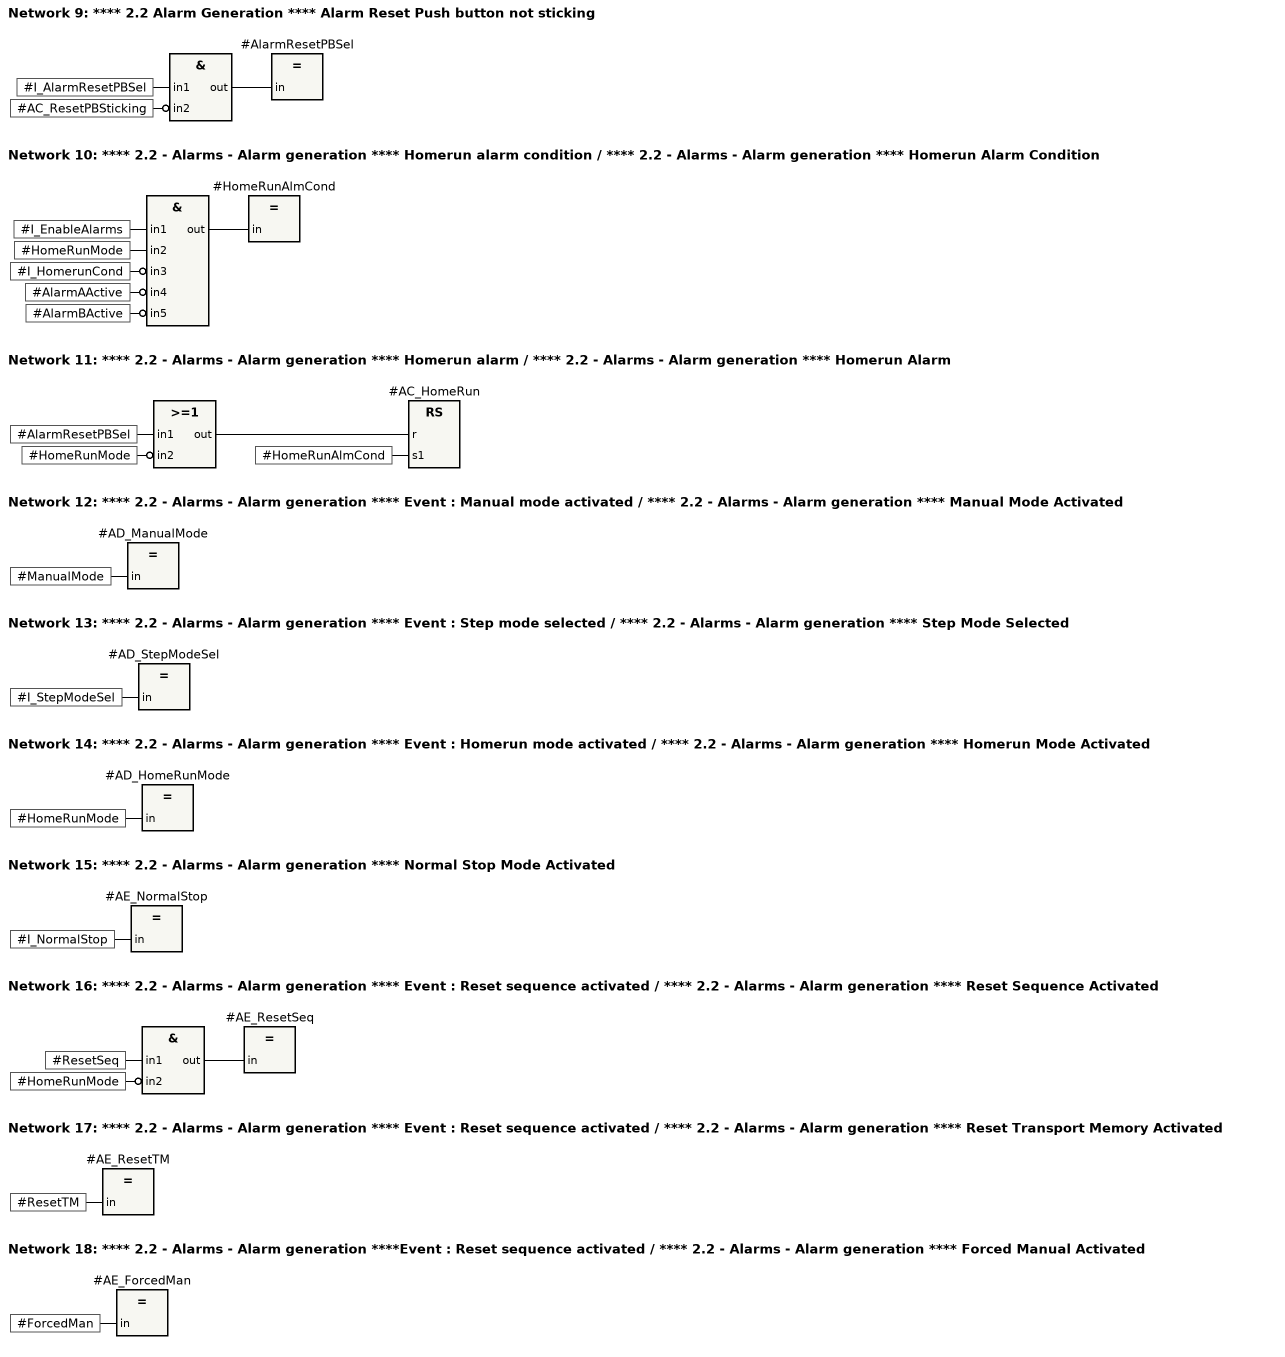
   #AlarmResetPBSel := #I_AlarmResetPBSel AND NOT #AC_ResetPBSticking;
END_REGION

REGION Network 10: **** 2.2 - Alarms - Alarm generation **** Homerun alarm condition / **** 2.2 - Alarms - Alarm generation **** Homerun Alarm Condition
   // Homerun alarm condition
   #HomeRunAlmCond := #I_EnableAlarms AND #HomeRunMode AND NOT #I_HomerunCond AND NOT #AlarmAActive AND NOT #AlarmBActive;
END_REGION

REGION Network 11: **** 2.2 - Alarms - Alarm generation **** Homerun alarm / **** 2.2 - Alarms - Alarm generation **** Homerun Alarm
   // Homerun alarm
   IF #AlarmResetPBSel OR NOT #HomeRunMode THEN
       #AC_HomeRun := FALSE;   // RS flip-flop
   END_IF;
   IF #HomeRunAlmCond THEN #AC_HomeRun := TRUE; END_IF;
END_REGION

REGION Network 12: **** 2.2 - Alarms - Alarm generation **** Event : Manual mode activated / **** 2.2 - Alarms - Alarm generation **** Manual Mode Activated
   // Event : Manual mode activated / Event : Manual Mode activated
   #AD_ManualMode := #ManualMode;
END_REGION

REGION Network 13: **** 2.2 - Alarms - Alarm generation **** Event : Step mode selected / **** 2.2 - Alarms - Alarm generation **** Step Mode Selected
   // Event : Step mode selected / Event : Step Mode selected
   #AD_StepModeSel := #I_StepModeSel;
END_REGION

REGION Network 14: **** 2.2 - Alarms - Alarm generation **** Event : Homerun mode activated / **** 2.2 - Alarms - Alarm generation **** Homerun Mode Activated
   // Event : Homerun mode activated / Event : Homerun Mode activated
   #AD_HomeRunMode := #HomeRunMode;
END_REGION

REGION Network 15: **** 2.2 - Alarms - Alarm generation **** Normal Stop Mode Activated
   // Event : Normal Stop Mode activated
   #AE_NormalStop := #I_NormalStop;
END_REGION

REGION Network 16: **** 2.2 - Alarms - Alarm generation **** Event : Reset sequence activated / **** 2.2 - Alarms - Alarm generation **** Reset Sequence Activated
   // Event : Reset sequence activated
   #AE_ResetSeq := #ResetSeq AND NOT #HomeRunMode;
END_REGION

REGION Network 17: **** 2.2 - Alarms - Alarm generation **** Event : Reset sequence activated / **** 2.2 - Alarms - Alarm generation **** Reset Transport Memory Activated
   // Event : Reset sequence activated / Event : Reset transport memory activated
   #AE_ResetTM := #ResetTM;
END_REGION

REGION Network 18: **** 2.2 - Alarms - Alarm generation ****Event : Reset sequence activated / **** 2.2 - Alarms - Alarm generation **** Forced Manual Activated
   // Event : Reset sequence activated / Event : Forced manual activated
   #AE_ForcedMan := #ForcedMan;
END_REGION

REGION Network 19: **** 2.2 - Alarms - Alarm generation **** Auto selected, but not started / **** 2.2 - Alarms - Alarm generation **** Auto Selected, But not Started
   // Auto selected, but not started
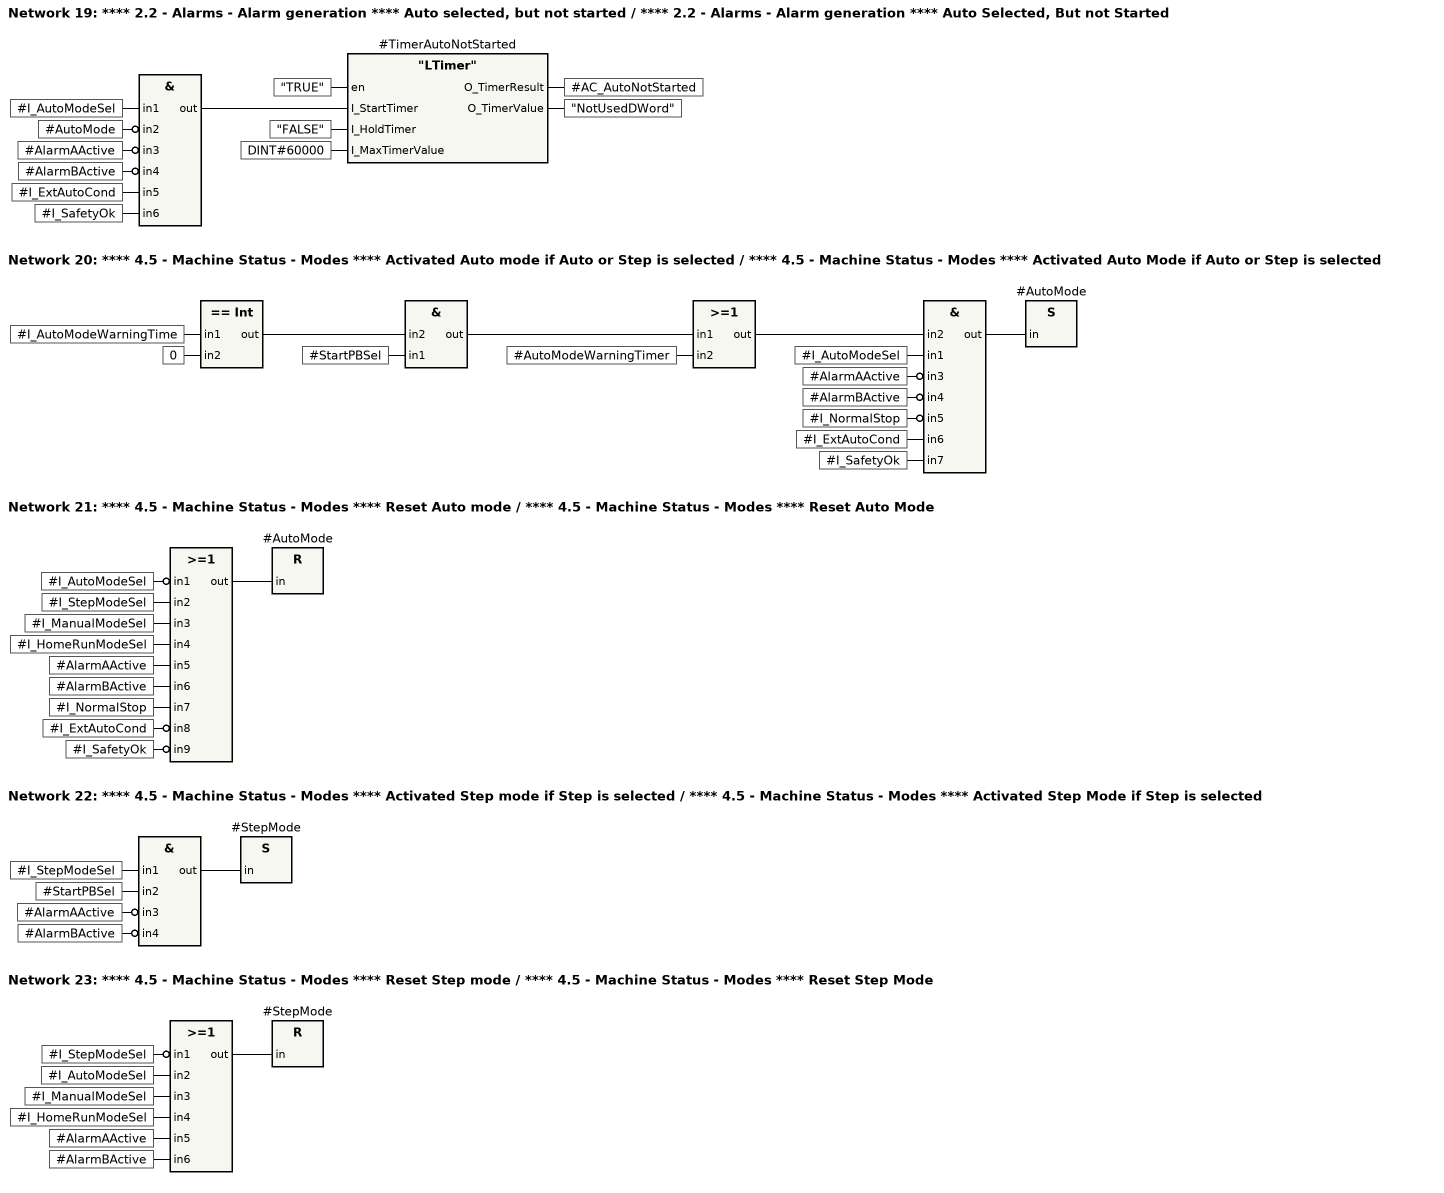
   IF "TRUE" THEN
       #TimerAutoNotStarted(I_StartTimer := #I_AutoModeSel AND NOT #AutoMode AND NOT #AlarmAActive AND NOT #AlarmBActive AND #I_ExtAutoCond AND #I_SafetyOk,   // "LTimer"
                            I_HoldTimer := "FALSE",
                            I_MaxTimerValue := DINT#60000,
                            O_TimerResult => #AC_AutoNotStarted,
                            O_TimerValue => "NotUsedDWord");
   END_IF;
END_REGION

REGION Network 20: **** 4.5 - Machine Status - Modes **** Activated Auto mode if Auto or Step is selected / **** 4.5 - Machine Status - Modes **** Activated Auto Mode if Auto or Step is selected
   // Activated Auto mode if Auto or Step is selected / Activated Auto Mode if Auto or Step is selected
   IF (((#I_AutoModeWarningTime = 0) AND #StartPBSel) OR #AutoModeWarningTimer) AND #I_AutoModeSel AND NOT #AlarmAActive AND NOT #AlarmBActive AND NOT #I_NormalStop AND #I_ExtAutoCond AND #I_SafetyOk THEN
       #AutoMode := TRUE;
   END_IF;
END_REGION

REGION Network 21: **** 4.5 - Machine Status - Modes **** Reset Auto mode / **** 4.5 - Machine Status - Modes **** Reset Auto Mode
   // Reset Auto mode / Reset Auto Mode
   IF NOT #I_AutoModeSel OR #I_StepModeSel OR #I_ManualModeSel OR #I_HomeRunModeSel OR #AlarmAActive OR #AlarmBActive OR #I_NormalStop OR NOT #I_ExtAutoCond OR NOT #I_SafetyOk THEN
       #AutoMode := FALSE;
   END_IF;
END_REGION

REGION Network 22: **** 4.5 - Machine Status - Modes **** Activated Step mode if Step is selected / **** 4.5 - Machine Status - Modes **** Activated Step Mode if Step is selected
   // Activated Step mode if Step is selected / Activated Step Mode if Step is selected
   IF #I_StepModeSel AND #StartPBSel AND NOT #AlarmAActive AND NOT #AlarmBActive THEN
       #StepMode := TRUE;
   END_IF;
END_REGION

REGION Network 23: **** 4.5 - Machine Status - Modes **** Reset Step mode / **** 4.5 - Machine Status - Modes **** Reset Step Mode
   // Reset Step mode / Reset Step Mode
   IF NOT #I_StepModeSel OR #I_AutoModeSel OR #I_ManualModeSel OR #I_HomeRunModeSel OR #AlarmAActive OR #AlarmBActive THEN
       #StepMode := FALSE;
   END_IF;
END_REGION

REGION Network 24: **** 4.5 - Machine Status - Modes **** Activate Homerun mode if all robots are out of station / **** 4.5 - Machine Status - Modes **** Activate Homerun Mode if all robots are out of station
   // Activate Homerun mode if all robots are out of station / Activate Homerun Mode if all robots are out of station
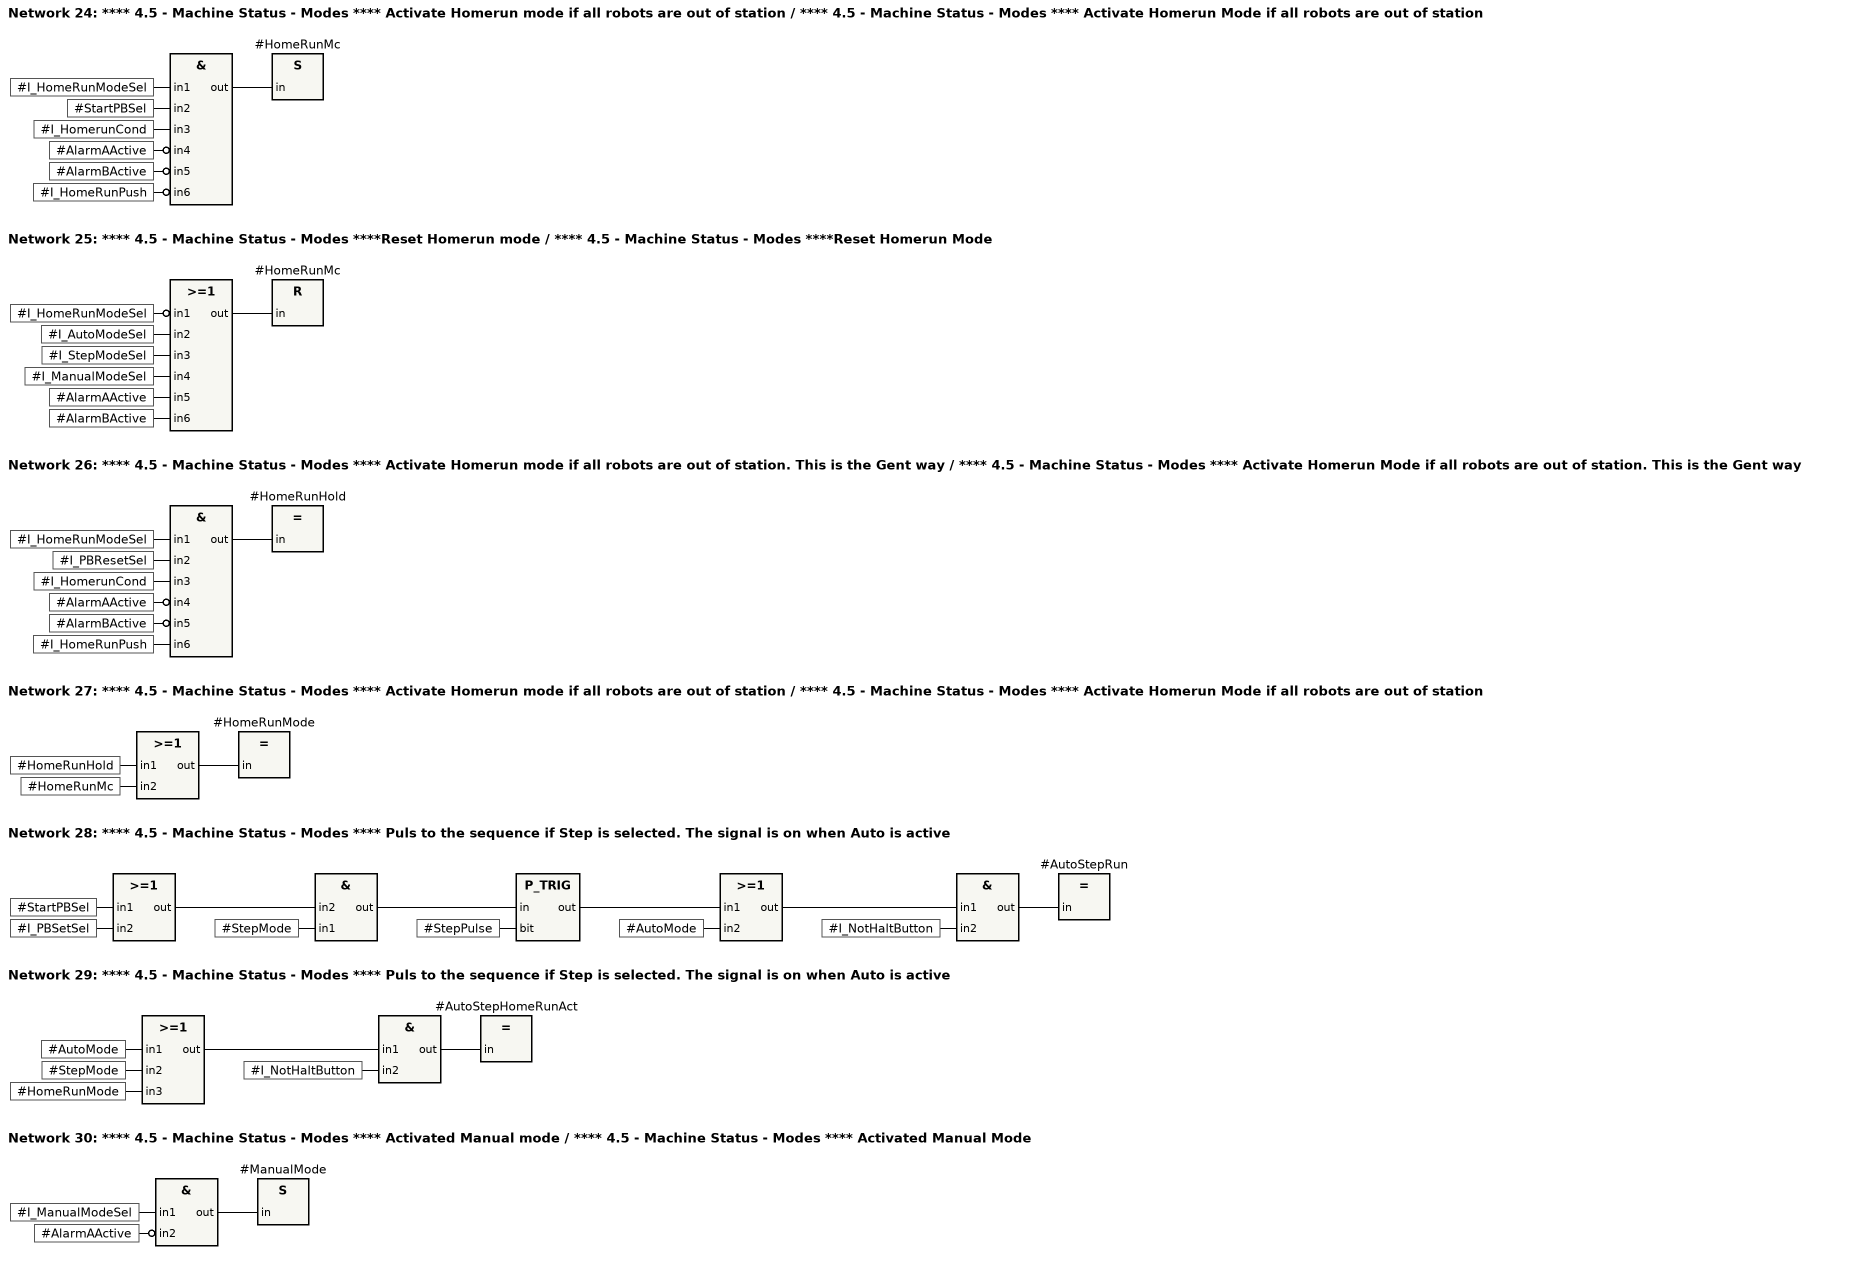
   IF #I_HomeRunModeSel AND #StartPBSel AND #I_HomerunCond AND NOT #AlarmAActive AND NOT #AlarmBActive AND NOT #I_HomeRunPush THEN
       #HomeRunMc := TRUE;
   END_IF;
END_REGION

REGION Network 25: **** 4.5 - Machine Status - Modes ****Reset Homerun mode / **** 4.5 - Machine Status - Modes ****Reset Homerun Mode
   // Reset Homerun mode / Reset Homerun Mode
   IF NOT #I_HomeRunModeSel OR #I_AutoModeSel OR #I_StepModeSel OR #I_ManualModeSel OR #AlarmAActive OR #AlarmBActive THEN
       #HomeRunMc := FALSE;
   END_IF;
END_REGION

REGION Network 26: **** 4.5 - Machine Status - Modes **** Activate Homerun mode if all robots are out of station. This is the Gent way / **** 4.5 - Machine Status - Modes **** Activate Homerun Mode if all robots are out of station. This is the Gent way
   // Activate Homerun mode if all robots are out of station. This is the Gent way 
   // there the reset pushbutton have to be pressed during the complete homerun.
   // Activate Homerun Mode if all robots are out of station. This is the Gent way 
   // there the reset pushbutton have to be pressed during the complete homerun.
   #HomeRunHold := #I_HomeRunModeSel AND #I_PBResetSel AND #I_HomerunCond AND NOT #AlarmAActive AND NOT #AlarmBActive AND #I_HomeRunPush;
END_REGION

REGION Network 27: **** 4.5 - Machine Status - Modes **** Activate Homerun mode if all robots are out of station / **** 4.5 - Machine Status - Modes **** Activate Homerun Mode if all robots are out of station
   // Activate Homerun mode if all robots are out of station. / Activate Homerun Mode if all robots are out of station.
   #HomeRunMode := #HomeRunHold OR #HomeRunMc;
END_REGION

REGION Network 28: **** 4.5 - Machine Status - Modes **** Puls to the sequence if Step is selected. The signal is on when Auto is active
   // Puls to the sequence if Step is selected. The signal is on when Auto is active.
   #_w1 := (#StartPBSel OR #I_PBSetSel) AND #StepMode;
   #_w2 := #_w1 AND NOT #StepPulse;   // rising edge
   #StepPulse := #_w1;
   #AutoStepRun := (#_w2 OR #AutoMode) AND #I_NotHaltButton;
END_REGION

REGION Network 29: **** 4.5 - Machine Status - Modes **** Puls to the sequence if Step is selected. The signal is on when Auto is active
   // Puls to the sequence if Step is selected. The signal is on when Auto is active.
   #AutoStepHomeRunAct := (#AutoMode OR #StepMode OR #HomeRunMode) AND #I_NotHaltButton;
END_REGION

REGION Network 30: **** 4.5 - Machine Status - Modes **** Activated Manual mode / **** 4.5 - Machine Status - Modes **** Activated Manual Mode
   // Activated Manual mode / Activated Manual Mode
   IF #I_ManualModeSel AND NOT #AlarmAActive THEN #ManualMode := TRUE; END_IF;
END_REGION

REGION Network 31: **** 4.5 - Machine Status - Modes **** Reset Manual mode / **** 4.5 - Machine Status - Modes **** Reset Manual Mode
   // Reset Manual mode / Reset Manual Mode
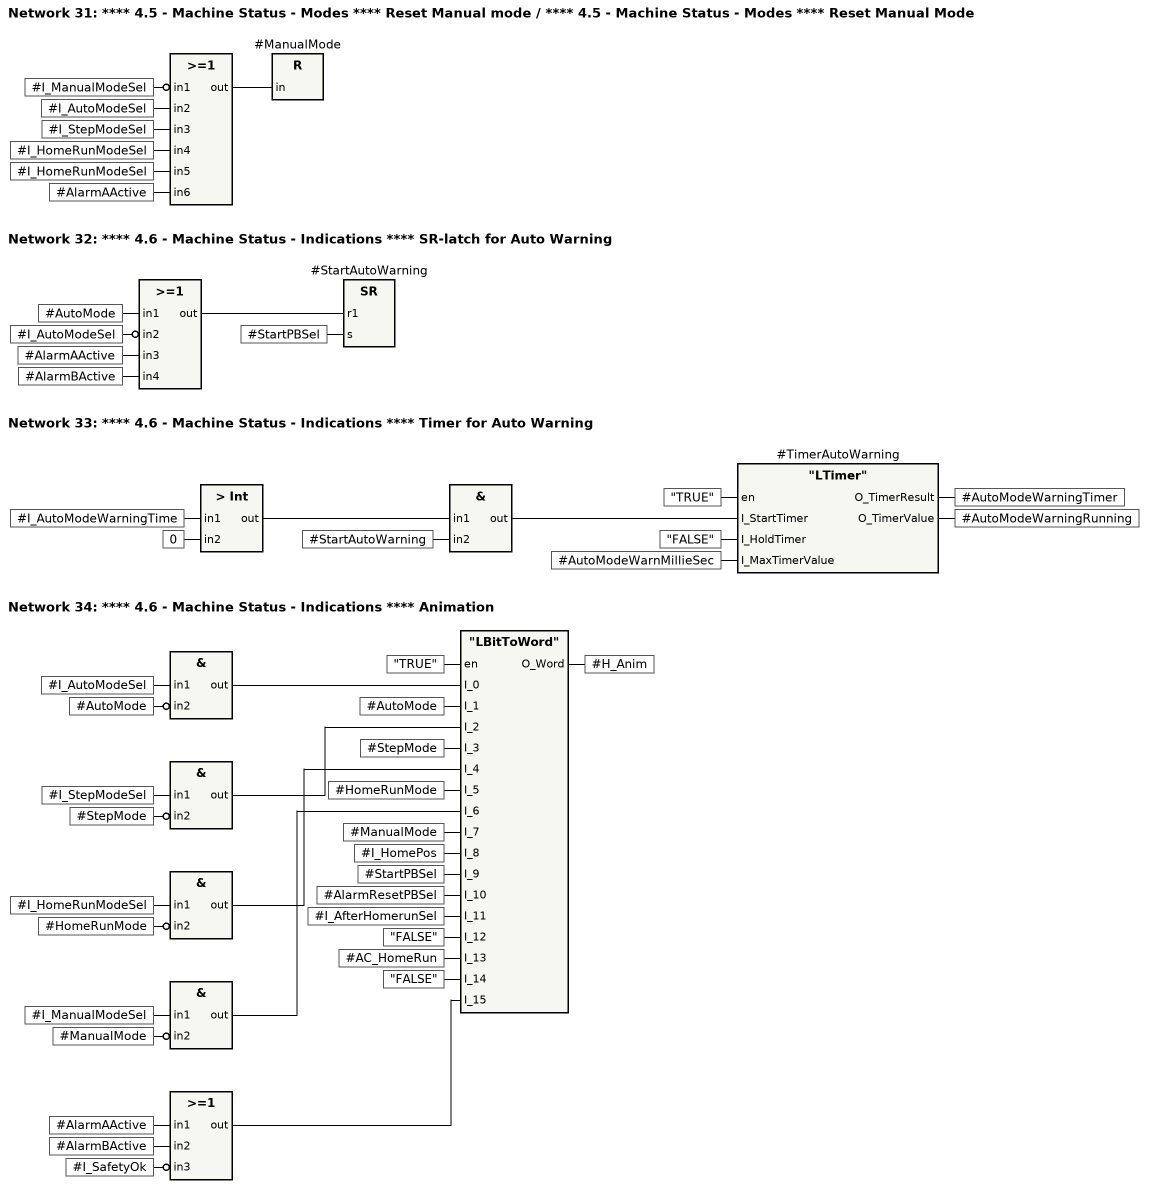
   IF NOT #I_ManualModeSel OR #I_AutoModeSel OR #I_StepModeSel OR #I_HomeRunModeSel OR #I_HomeRunModeSel OR #AlarmAActive THEN
       #ManualMode := FALSE;
   END_IF;
END_REGION

REGION Network 32: **** 4.6 - Machine Status - Indications **** SR-latch for Auto Warning
   // SR-latch for Auto Warning
   IF #StartPBSel THEN
       #StartAutoWarning := TRUE;   // SR flip-flop
   END_IF;
   IF #AutoMode OR NOT #I_AutoModeSel OR #AlarmAActive OR #AlarmBActive THEN
       #StartAutoWarning := FALSE;
   END_IF;
END_REGION

REGION Network 33: **** 4.6 - Machine Status - Indications **** Timer for Auto Warning
   // Timer for Auto Warning
   IF "TRUE" THEN
       #TimerAutoWarning(I_StartTimer := (#I_AutoModeWarningTime > 0) AND #StartAutoWarning,   // "LTimer"
                         I_HoldTimer := "FALSE",
                         I_MaxTimerValue := #AutoModeWarnMillieSec,
                         O_TimerResult => #AutoModeWarningTimer,
                         O_TimerValue => #AutoModeWarningRunning);
   END_IF;
END_REGION

REGION Network 34: **** 4.6 - Machine Status - Indications **** Animation
   // Animation
   IF "TRUE" THEN
       "LBitToWord"(I_0 := #I_AutoModeSel AND NOT #AutoMode,
                    I_1 := #AutoMode,
                    I_2 := #I_StepModeSel AND NOT #StepMode,
                    I_3 := #StepMode,
                    I_4 := #I_HomeRunModeSel AND NOT #HomeRunMode,
                    I_5 := #HomeRunMode,
                    I_6 := #I_ManualModeSel AND NOT #ManualMode,
                    I_7 := #ManualMode,
                    I_8 := #I_HomePos,
                    I_9 := #StartPBSel,
                    I_10 := #AlarmResetPBSel,
                    I_11 := #I_AfterHomerunSel,
                    I_12 := "FALSE",
                    I_13 := #AC_HomeRun,
                    I_14 := "FALSE",
                    I_15 := #AlarmAActive OR #AlarmBActive OR NOT #I_SafetyOk,
                    O_Word => #H_Anim);
   END_IF;
END_REGION

REGION Network 35: **** 4.6 - Machine Status - Indications **** Animation2
   // Animation
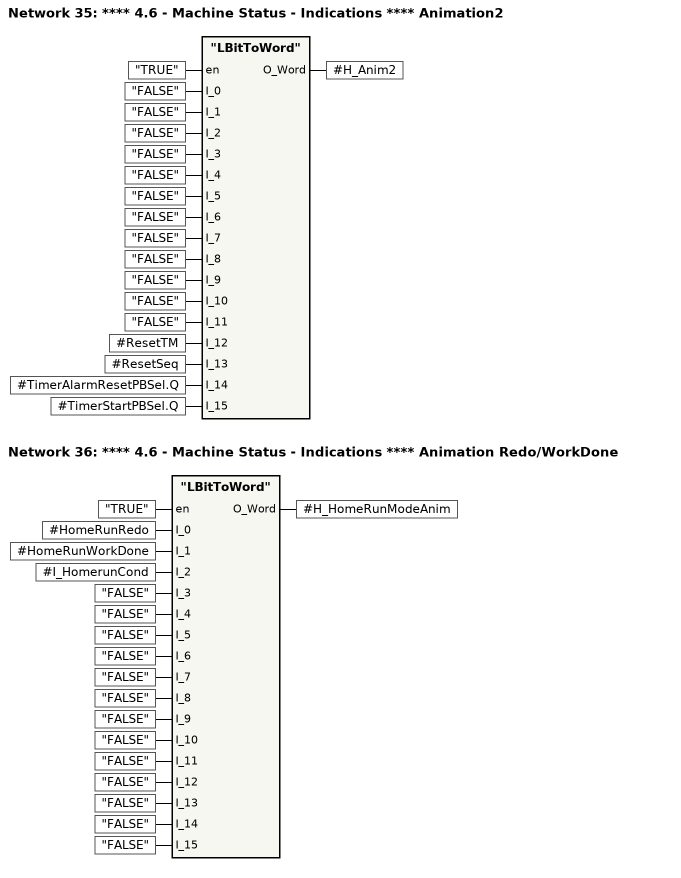
   IF "TRUE" THEN
       "LBitToWord"(I_0 := "FALSE",
                    I_1 := "FALSE",
                    I_2 := "FALSE",
                    I_3 := "FALSE",
                    I_4 := "FALSE",
                    I_5 := "FALSE",
                    I_6 := "FALSE",
                    I_7 := "FALSE",
                    I_8 := "FALSE",
                    I_9 := "FALSE",
                    I_10 := "FALSE",
                    I_11 := "FALSE",
                    I_12 := #ResetTM,
                    I_13 := #ResetSeq,
                    I_14 := #TimerAlarmResetPBSel.Q,
                    I_15 := #TimerStartPBSel.Q,
                    O_Word => #H_Anim2);
   END_IF;
END_REGION

REGION Network 36: **** 4.6 - Machine Status - Indications **** Animation Redo/WorkDone
   // Animation Redo/WorkDone
   IF "TRUE" THEN
       "LBitToWord"(I_0 := #HomeRunRedo,
                    I_1 := #HomeRunWorkDone,
                    I_2 := #I_HomerunCond,
                    I_3 := "FALSE",
                    I_4 := "FALSE",
                    I_5 := "FALSE",
                    I_6 := "FALSE",
                    I_7 := "FALSE",
                    I_8 := "FALSE",
                    I_9 := "FALSE",
                    I_10 := "FALSE",
                    I_11 := "FALSE",
                    I_12 := "FALSE",
                    I_13 := "FALSE",
                    I_14 := "FALSE",
                    I_15 := "FALSE",
                    O_Word => #H_HomeRunModeAnim);
   END_IF;
END_REGION

REGION Network 37: **** 4.6 - Machine Status - Indications **** Animation HMI LED
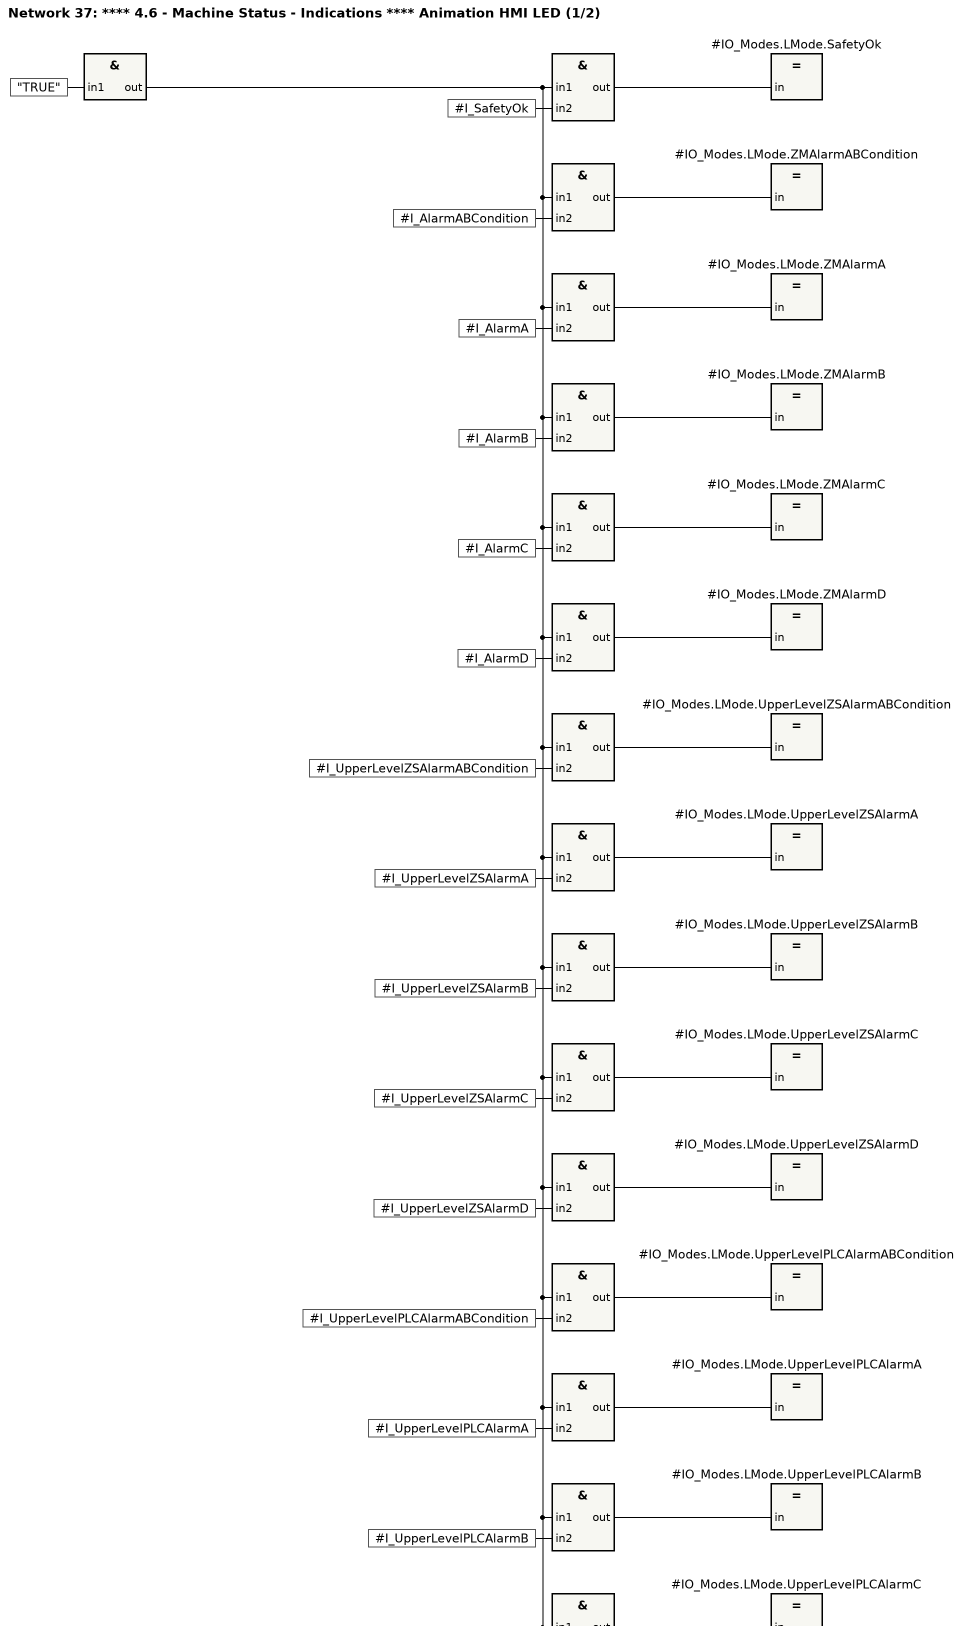
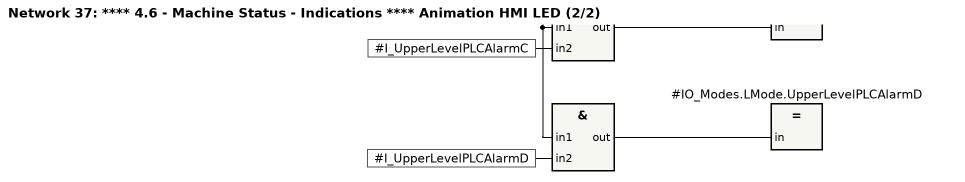
   #IO_Modes.LMode.SafetyOk := "TRUE" AND #I_SafetyOk;
   #IO_Modes.LMode.ZMAlarmABCondition := "TRUE" AND #I_AlarmABCondition;
   #IO_Modes.LMode.ZMAlarmA := "TRUE" AND #I_AlarmA;
   #IO_Modes.LMode.ZMAlarmB := "TRUE" AND #I_AlarmB;
   #IO_Modes.LMode.ZMAlarmC := "TRUE" AND #I_AlarmC;
   #IO_Modes.LMode.ZMAlarmD := "TRUE" AND #I_AlarmD;
   #IO_Modes.LMode.UpperLevelZSAlarmABCondition := "TRUE" AND #I_UpperLevelZSAlarmABCondition;
   #IO_Modes.LMode.UpperLevelZSAlarmA := "TRUE" AND #I_UpperLevelZSAlarmA;
   #IO_Modes.LMode.UpperLevelZSAlarmB := "TRUE" AND #I_UpperLevelZSAlarmB;
   #IO_Modes.LMode.UpperLevelZSAlarmC := "TRUE" AND #I_UpperLevelZSAlarmC;
   #IO_Modes.LMode.UpperLevelZSAlarmD := "TRUE" AND #I_UpperLevelZSAlarmD;
   #IO_Modes.LMode.UpperLevelPLCAlarmABCondition := "TRUE" AND #I_UpperLevelPLCAlarmABCondition;
   #IO_Modes.LMode.UpperLevelPLCAlarmA := "TRUE" AND #I_UpperLevelPLCAlarmA;
   #IO_Modes.LMode.UpperLevelPLCAlarmB := "TRUE" AND #I_UpperLevelPLCAlarmB;
   #IO_Modes.LMode.UpperLevelPLCAlarmC := "TRUE" AND #I_UpperLevelPLCAlarmC;
   #IO_Modes.LMode.UpperLevelPLCAlarmD := "TRUE" AND #I_UpperLevelPLCAlarmD;
END_REGION

REGION Network 38: **** 5.2 - Equations - Flow **** Manual mode is active and the Forced key switch is activated / **** 5.2 - Equations - Flow **** Manual Mode is active and the Forced key switch is activated
   // Manual mode is active and the Forced key switch is activated / Manual Mode is active and the Forced key switch is activated
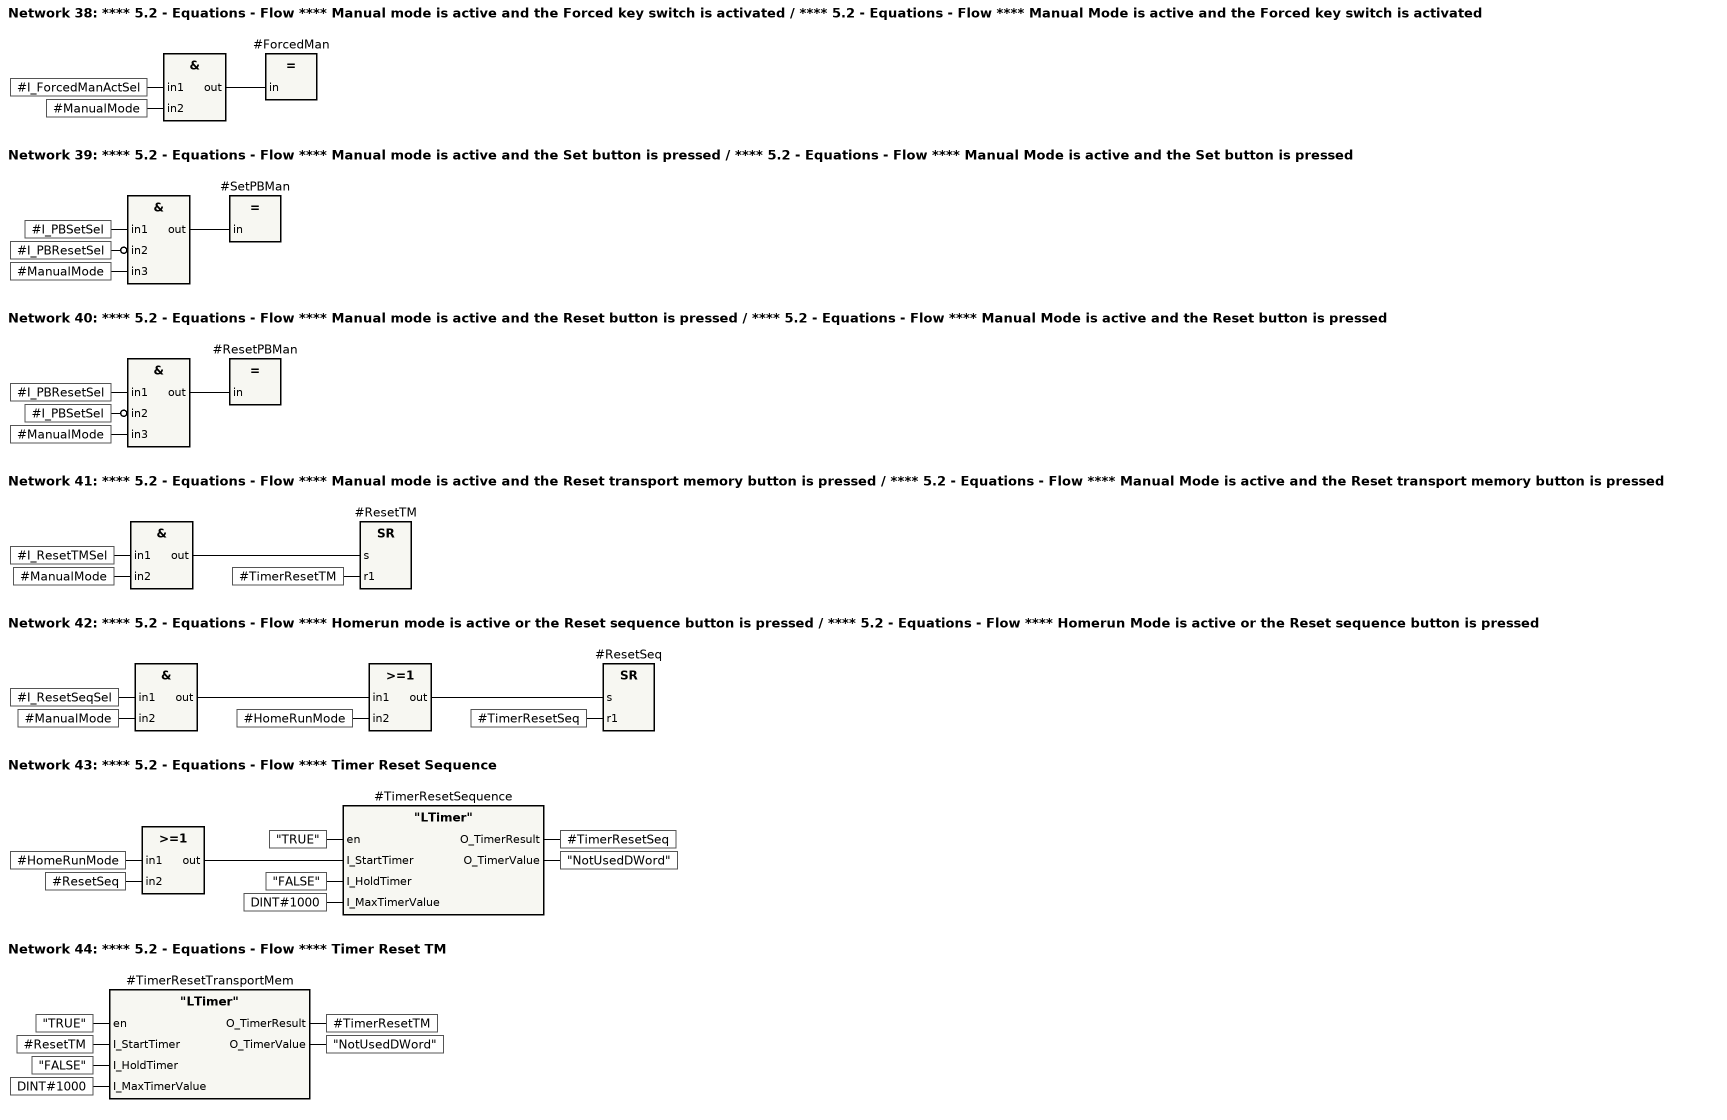
   #ForcedMan := #I_ForcedManActSel AND #ManualMode;
END_REGION

REGION Network 39: **** 5.2 - Equations - Flow **** Manual mode is active and the Set button is pressed / **** 5.2 - Equations - Flow **** Manual Mode is active and the Set button is pressed
   // Manual mode is active and the Set button is pressed / Manual Mode is active and the Set button is pressed
   #SetPBMan := #I_PBSetSel AND NOT #I_PBResetSel AND #ManualMode;
END_REGION

REGION Network 40: **** 5.2 - Equations - Flow **** Manual mode is active and the Reset button is pressed / **** 5.2 - Equations - Flow **** Manual Mode is active and the Reset button is pressed
   // Manual mode is active and the Reset button is pressed / Manual Mode is active and the Reset button is pressed
   #ResetPBMan := #I_PBResetSel AND NOT #I_PBSetSel AND #ManualMode;
END_REGION

REGION Network 41: **** 5.2 - Equations - Flow **** Manual mode is active and the Reset transport memory button is pressed / **** 5.2 - Equations - Flow **** Manual Mode is active and the Reset transport memory button is pressed
   // Manual mode is active and the Reset transport memory button is pressed / Manual Mode is active and the Reset transport memory button is pressed
   IF #I_ResetTMSel AND #ManualMode THEN
       #ResetTM := TRUE;   // SR flip-flop
   END_IF;
   IF #TimerResetTM THEN #ResetTM := FALSE; END_IF;
END_REGION

REGION Network 42: **** 5.2 - Equations - Flow **** Homerun mode is active or the Reset sequence button is pressed / **** 5.2 - Equations - Flow **** Homerun Mode is active or the Reset sequence button is pressed
   // Homerun mode is active or the Reset sequence button is pressed / Homerun Mode is active or the Reset sequence button is pressed
   IF (#I_ResetSeqSel AND #ManualMode) OR #HomeRunMode THEN
       #ResetSeq := TRUE;   // SR flip-flop
   END_IF;
   IF #TimerResetSeq THEN #ResetSeq := FALSE; END_IF;
END_REGION

REGION Network 43: **** 5.2 - Equations - Flow **** Timer Reset Sequence
   // Timer Reset Sequence
   IF "TRUE" THEN
       #TimerResetSequence(I_StartTimer := #HomeRunMode OR #ResetSeq,   // "LTimer"
                           I_HoldTimer := "FALSE",
                           I_MaxTimerValue := DINT#1000,
                           O_TimerResult => #TimerResetSeq,
                           O_TimerValue => "NotUsedDWord");
   END_IF;
END_REGION

REGION Network 44: **** 5.2 - Equations - Flow **** Timer Reset TM
   // Timer Reset TM
   IF "TRUE" THEN
       #TimerResetTransportMem(I_StartTimer := #ResetTM,   // "LTimer"
                               I_HoldTimer := "FALSE",
                               I_MaxTimerValue := DINT#1000,
                               O_TimerResult => #TimerResetTM,
                               O_TimerValue => "NotUsedDWord");
   END_IF;
END_REGION

REGION Network 45: **** 5.2 - Equations - Flow **** Redo after homerun
   // Redo after homerun
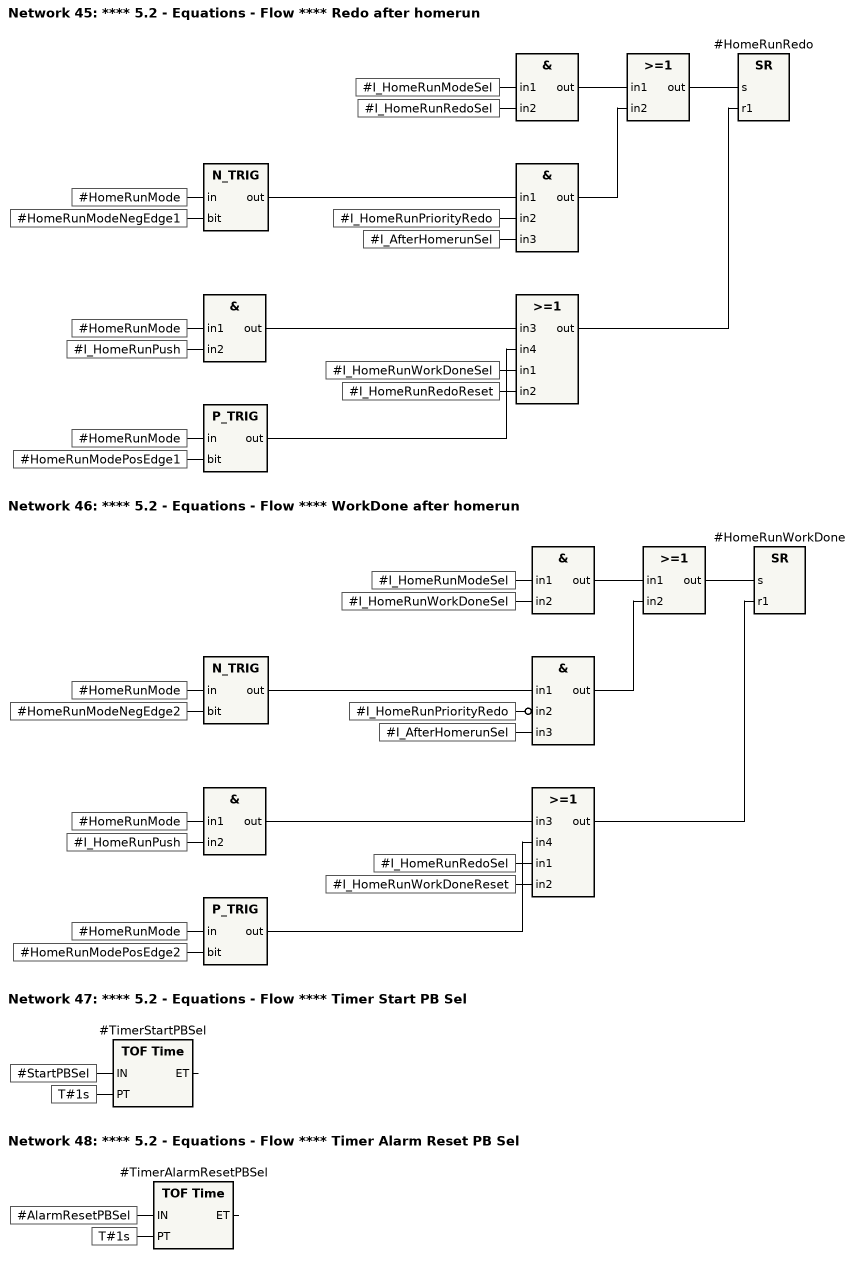
   #_w1 := NOT #HomeRunMode AND #HomeRunModeNegEdge1;   // falling edge
   #HomeRunModeNegEdge1 := #HomeRunMode;
   #_w2 := #HomeRunMode AND NOT #HomeRunModePosEdge1;   // rising edge
   #HomeRunModePosEdge1 := #HomeRunMode;
   IF (#I_HomeRunModeSel AND #I_HomeRunRedoSel) OR (#_w1 AND #I_HomeRunPriorityRedo AND #I_AfterHomerunSel) THEN
       #HomeRunRedo := TRUE;   // SR flip-flop
   END_IF;
   IF (#HomeRunMode AND #I_HomeRunPush) OR #_w2 OR #I_HomeRunWorkDoneSel OR #I_HomeRunRedoReset THEN
       #HomeRunRedo := FALSE;
   END_IF;
END_REGION

REGION Network 46: **** 5.2 - Equations - Flow **** WorkDone after homerun
   // WorkDone after homerun
   #_w1 := NOT #HomeRunMode AND #HomeRunModeNegEdge2;   // falling edge
   #HomeRunModeNegEdge2 := #HomeRunMode;
   #_w2 := #HomeRunMode AND NOT #HomeRunModePosEdge2;   // rising edge
   #HomeRunModePosEdge2 := #HomeRunMode;
   IF (#I_HomeRunModeSel AND #I_HomeRunWorkDoneSel) OR (#_w1 AND NOT #I_HomeRunPriorityRedo AND #I_AfterHomerunSel) THEN
       #HomeRunWorkDone := TRUE;   // SR flip-flop
   END_IF;
   IF (#HomeRunMode AND #I_HomeRunPush) OR #_w2 OR #I_HomeRunRedoSel OR #I_HomeRunWorkDoneReset THEN
       #HomeRunWorkDone := FALSE;
   END_IF;
END_REGION

REGION Network 47: **** 5.2 - Equations - Flow **** Timer Start PB Sel
   // Timer Start PB Sel
   #TimerStartPBSel(IN := #StartPBSel, PT := T#1s);   // TOF
END_REGION

REGION Network 48: **** 5.2 - Equations - Flow **** Timer Alarm Reset PB Sel
   // Timer Alarm Reset PB Sel
   #TimerAlarmResetPBSel(IN := #AlarmResetPBSel, PT := T#1s);   // TOF
END_REGION

REGION Network 49: **** 8 - Outputs **** Set the different bits in the Mode register
   // Set the different bits in the Mode register
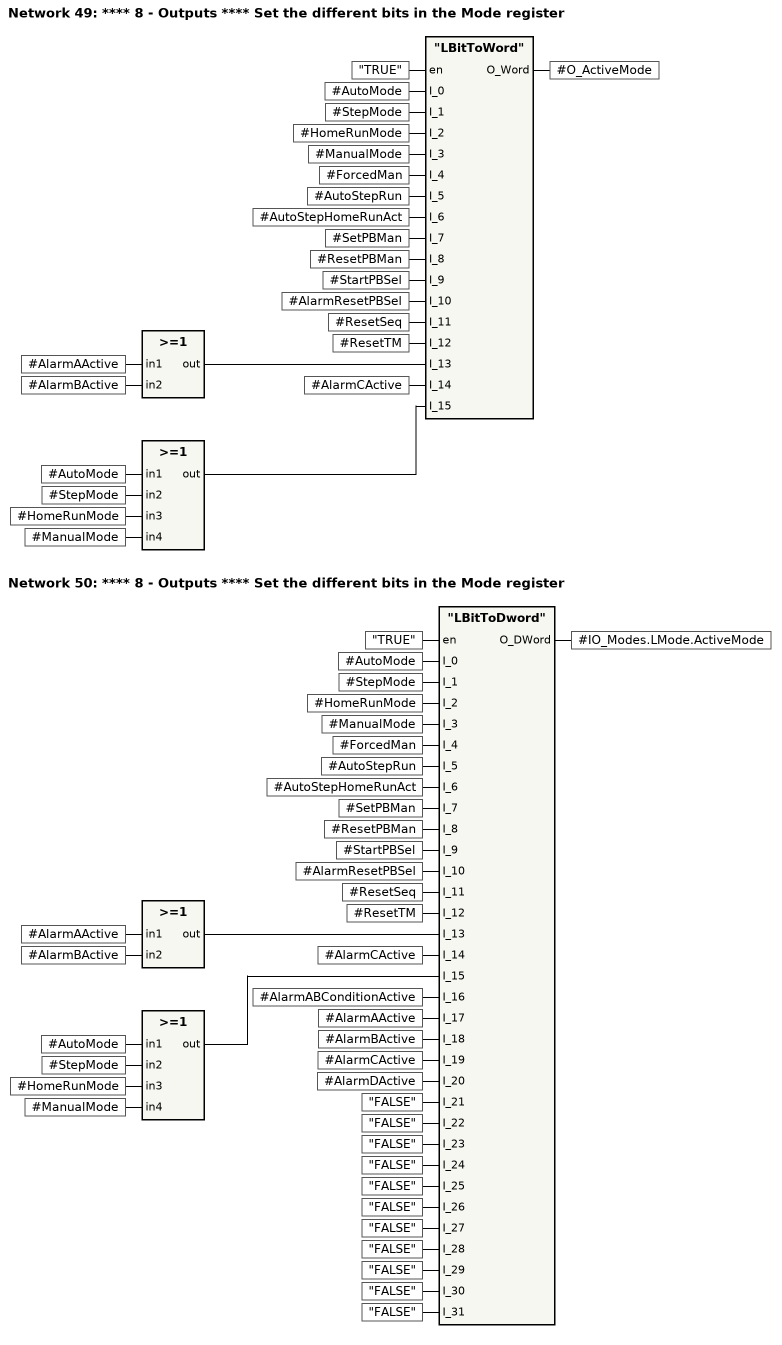
   IF "TRUE" THEN
       "LBitToWord"(I_0 := #AutoMode,
                    I_1 := #StepMode,
                    I_2 := #HomeRunMode,
                    I_3 := #ManualMode,
                    I_4 := #ForcedMan,
                    I_5 := #AutoStepRun,
                    I_6 := #AutoStepHomeRunAct,
                    I_7 := #SetPBMan,
                    I_8 := #ResetPBMan,
                    I_9 := #StartPBSel,
                    I_10 := #AlarmResetPBSel,
                    I_11 := #ResetSeq,
                    I_12 := #ResetTM,
                    I_13 := #AlarmAActive OR #AlarmBActive,
                    I_14 := #AlarmCActive,
                    I_15 := #AutoMode OR #StepMode OR #HomeRunMode OR #ManualMode,
                    O_Word => #O_ActiveMode);
   END_IF;
END_REGION

REGION Network 50: **** 8 - Outputs **** Set the different bits in the Mode register
   // Set the different bits in the Mode register
   IF "TRUE" THEN
       "LBitToDword"(I_0 := #AutoMode,
                     I_1 := #StepMode,
                     I_2 := #HomeRunMode,
                     I_3 := #ManualMode,
                     I_4 := #ForcedMan,
                     I_5 := #AutoStepRun,
                     I_6 := #AutoStepHomeRunAct,
                     I_7 := #SetPBMan,
                     I_8 := #ResetPBMan,
                     I_9 := #StartPBSel,
                     I_10 := #AlarmResetPBSel,
                     I_11 := #ResetSeq,
                     I_12 := #ResetTM,
                     I_13 := #AlarmAActive OR #AlarmBActive,
                     I_14 := #AlarmCActive,
                     I_15 := #AutoMode OR #StepMode OR #HomeRunMode OR #ManualMode,
                     I_16 := #AlarmABConditionActive,
                     I_17 := #AlarmAActive,
                     I_18 := #AlarmBActive,
                     I_19 := #AlarmCActive,
                     I_20 := #AlarmDActive,
                     I_21 := "FALSE",
                     I_22 := "FALSE",
                     I_23 := "FALSE",
                     I_24 := "FALSE",
                     I_25 := "FALSE",
                     I_26 := "FALSE",
                     I_27 := "FALSE",
                     I_28 := "FALSE",
                     I_29 := "FALSE",
                     I_30 := "FALSE",
                     I_31 := "FALSE",
                     O_DWord => #IO_Modes.LMode.ActiveMode);
   END_IF;
END_REGION

REGION Network 51: **** 8 - Outputs **** Set the different bits in the Mode register
   // Set the different bits in the Mode register
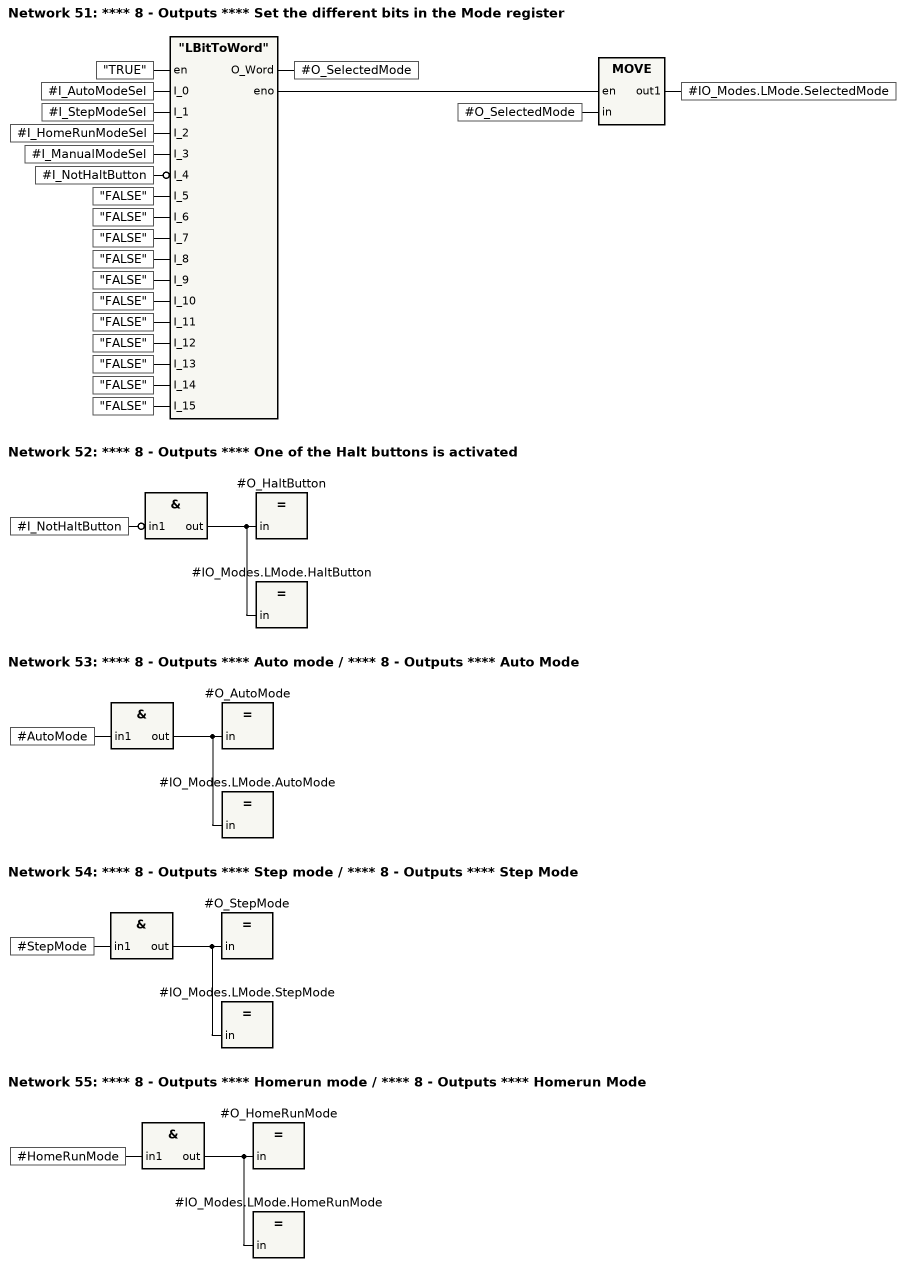
   "LBitToWord"(EN := "TRUE",
                I_0 := #I_AutoModeSel,
                I_1 := #I_StepModeSel,
                I_2 := #I_HomeRunModeSel,
                I_3 := #I_ManualModeSel,
                I_4 := NOT #I_NotHaltButton,
                I_5 := "FALSE",
                I_6 := "FALSE",
                I_7 := "FALSE",
                I_8 := "FALSE",
                I_9 := "FALSE",
                I_10 := "FALSE",
                I_11 := "FALSE",
                I_12 := "FALSE",
                I_13 := "FALSE",
                I_14 := "FALSE",
                I_15 := "FALSE",
                O_Word => #O_SelectedMode,
                ENO => #_w1);
   IF #_w1 THEN #IO_Modes.LMode.SelectedMode := #O_SelectedMode; END_IF;
END_REGION

REGION Network 52: **** 8 - Outputs **** One of the Halt buttons is activated
   // One of the Halt buttons is activated
   #O_HaltButton := NOT #I_NotHaltButton;
   #IO_Modes.LMode.HaltButton := NOT #I_NotHaltButton;
END_REGION

REGION Network 53: **** 8 - Outputs **** Auto mode / **** 8 - Outputs **** Auto Mode
   // Auto mode / Auto Mode
   #O_AutoMode := #AutoMode;
   #IO_Modes.LMode.AutoMode := #AutoMode;
END_REGION

REGION Network 54: **** 8 - Outputs **** Step mode / **** 8 - Outputs **** Step Mode
   // Step mode / Step Mode
   #O_StepMode := #StepMode;
   #IO_Modes.LMode.StepMode := #StepMode;
END_REGION

REGION Network 55: **** 8 - Outputs **** Homerun mode / **** 8 - Outputs **** Homerun Mode
   // Homerun mode / Homerun Mode
   #O_HomeRunMode := #HomeRunMode;
   #IO_Modes.LMode.HomeRunMode := #HomeRunMode;
END_REGION

REGION Network 56: **** 8 - Outputs **** Manual mode / **** 8 - Outputs **** Manual Mode
   // Manual mode / Manual Mode
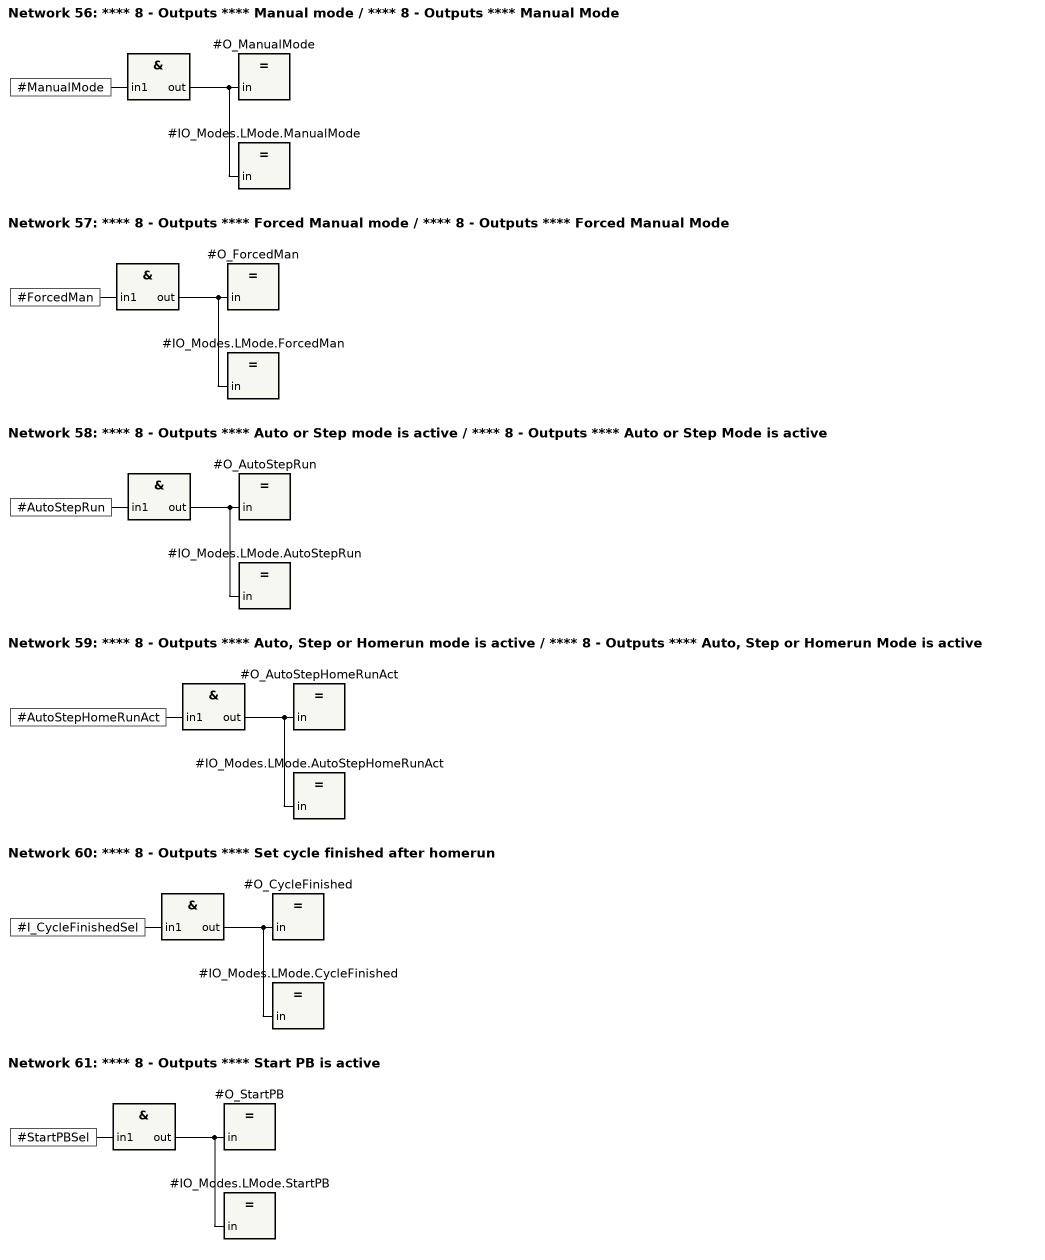
   #O_ManualMode := #ManualMode;
   #IO_Modes.LMode.ManualMode := #ManualMode;
END_REGION

REGION Network 57: **** 8 - Outputs **** Forced Manual mode / **** 8 - Outputs **** Forced Manual Mode
   // Forced Manual mode / Forced Manual Mode
   #O_ForcedMan := #ForcedMan;
   #IO_Modes.LMode.ForcedMan := #ForcedMan;
END_REGION

REGION Network 58: **** 8 - Outputs **** Auto or Step mode is active / **** 8 - Outputs **** Auto or Step Mode is active
   // Auto or Step mode is active / Auto or Step Mode is active
   #O_AutoStepRun := #AutoStepRun;
   #IO_Modes.LMode.AutoStepRun := #AutoStepRun;
END_REGION

REGION Network 59: **** 8 - Outputs **** Auto, Step or Homerun mode is active / **** 8 - Outputs **** Auto, Step or Homerun Mode is active
   // Auto, Step or Homerun mode is active / Auto, Step or Homerun Mode is active
   #O_AutoStepHomeRunAct := #AutoStepHomeRunAct;
   #IO_Modes.LMode.AutoStepHomeRunAct := #AutoStepHomeRunAct;
END_REGION

REGION Network 60: **** 8 - Outputs **** Set cycle finished after homerun
   // Set cycle finished after homerun
   #O_CycleFinished := #I_CycleFinishedSel;
   #IO_Modes.LMode.CycleFinished := #I_CycleFinishedSel;
END_REGION

REGION Network 61: **** 8 - Outputs **** Start PB is active
   // Start PB is active
   #O_StartPB := #StartPBSel;
   #IO_Modes.LMode.StartPB := #StartPBSel;
END_REGION

REGION Network 62: **** 8 - Outputs **** Alarm Reset PB is active
   // Alarm Reset PB is active
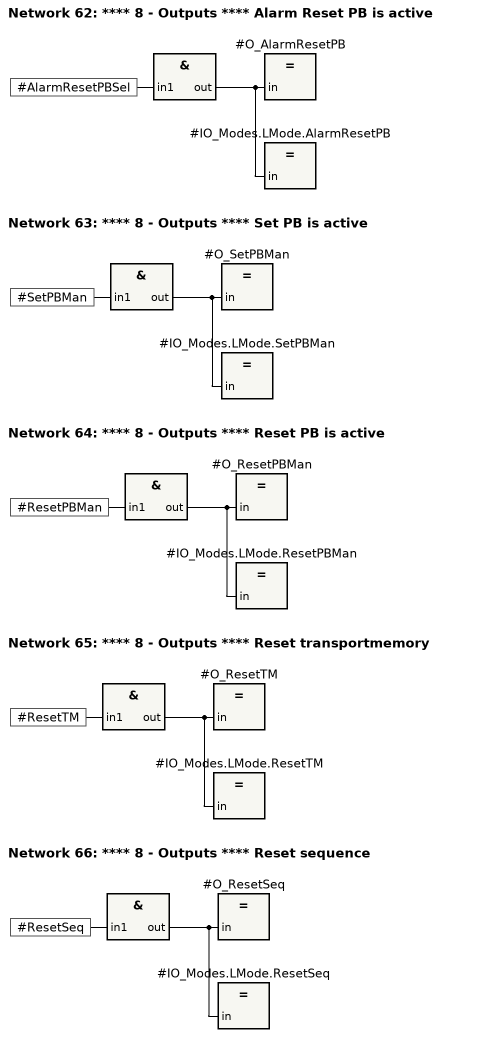
   #O_AlarmResetPB := #AlarmResetPBSel;
   #IO_Modes.LMode.AlarmResetPB := #AlarmResetPBSel;
END_REGION

REGION Network 63: **** 8 - Outputs **** Set PB is active
   // Set PB is active
   #O_SetPBMan := #SetPBMan;
   #IO_Modes.LMode.SetPBMan := #SetPBMan;
END_REGION

REGION Network 64: **** 8 - Outputs **** Reset PB is active
   // Reset PB is active
   #O_ResetPBMan := #ResetPBMan;
   #IO_Modes.LMode.ResetPBMan := #ResetPBMan;
END_REGION

REGION Network 65: **** 8 - Outputs **** Reset transportmemory
   // Reset transportmemory
   #O_ResetTM := #ResetTM;
   #IO_Modes.LMode.ResetTM := #ResetTM;
END_REGION

REGION Network 66: **** 8 - Outputs **** Reset sequence
   // Reset sequence
   #O_ResetSeq := #ResetSeq;
   #IO_Modes.LMode.ResetSeq := #ResetSeq;
END_REGION

REGION Network 67: **** 8 - Outputs **** Auto mode warning / **** 8 - Outputs **** Auto Mode warning
   // Auto mode warning / Auto Mode warning
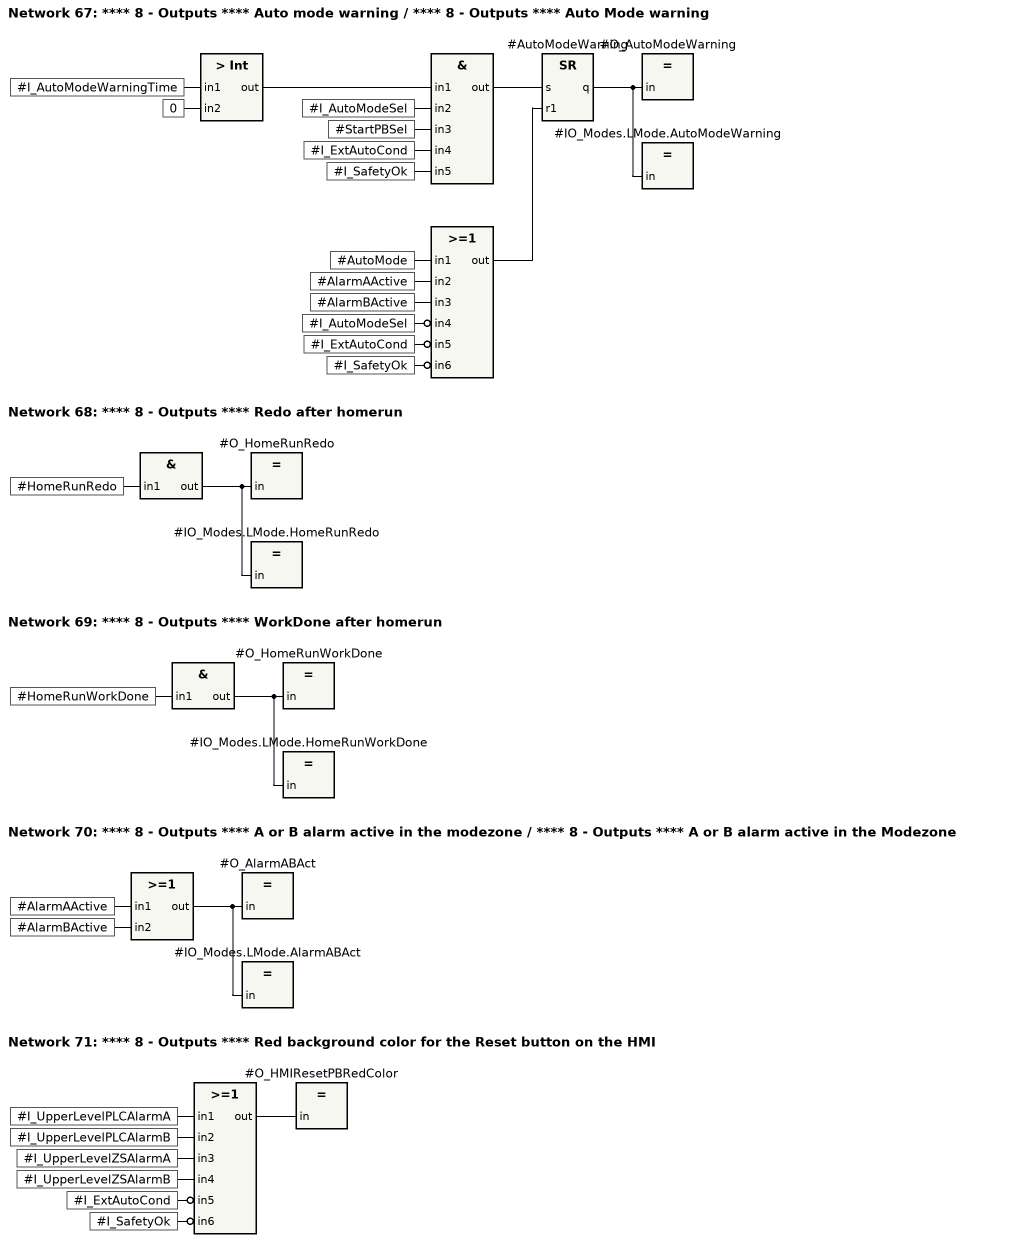
   IF (#I_AutoModeWarningTime > 0) AND #I_AutoModeSel AND #StartPBSel AND #I_ExtAutoCond AND #I_SafetyOk THEN
       #AutoModeWarning := TRUE;   // SR flip-flop
   END_IF;
   IF #AutoMode OR #AlarmAActive OR #AlarmBActive OR NOT #I_AutoModeSel OR NOT #I_ExtAutoCond OR NOT #I_SafetyOk THEN
       #AutoModeWarning := FALSE;
   END_IF;
   #O_AutoModeWarning := #AutoModeWarning;
   #IO_Modes.LMode.AutoModeWarning := #AutoModeWarning;
END_REGION

REGION Network 68: **** 8 - Outputs **** Redo after homerun
   // Redo after homerun
   #O_HomeRunRedo := #HomeRunRedo;
   #IO_Modes.LMode.HomeRunRedo := #HomeRunRedo;
END_REGION

REGION Network 69: **** 8 - Outputs **** WorkDone after homerun
   // WorkDone after homerun
   #O_HomeRunWorkDone := #HomeRunWorkDone;
   #IO_Modes.LMode.HomeRunWorkDone := #HomeRunWorkDone;
END_REGION

REGION Network 70: **** 8 - Outputs **** A or B alarm active in the modezone / **** 8 - Outputs **** A or B alarm active in the Modezone
   // A or B alarm active in the modezone / A or B alarm active in the Modezone
   #O_AlarmABAct := #AlarmAActive OR #AlarmBActive;
   #IO_Modes.LMode.AlarmABAct := #O_AlarmABAct;
END_REGION

REGION Network 71: **** 8 - Outputs **** Red background color for the Reset button on the HMI
   #O_HMIResetPBRedColor := #I_UpperLevelPLCAlarmA OR #I_UpperLevelPLCAlarmB OR #I_UpperLevelZSAlarmA OR #I_UpperLevelZSAlarmB OR NOT #I_ExtAutoCond OR NOT #I_SafetyOk;
END_REGION

REGION Network 72: **** 8 - Outputs **** Alarm AB condition
   // Alarm AB condition
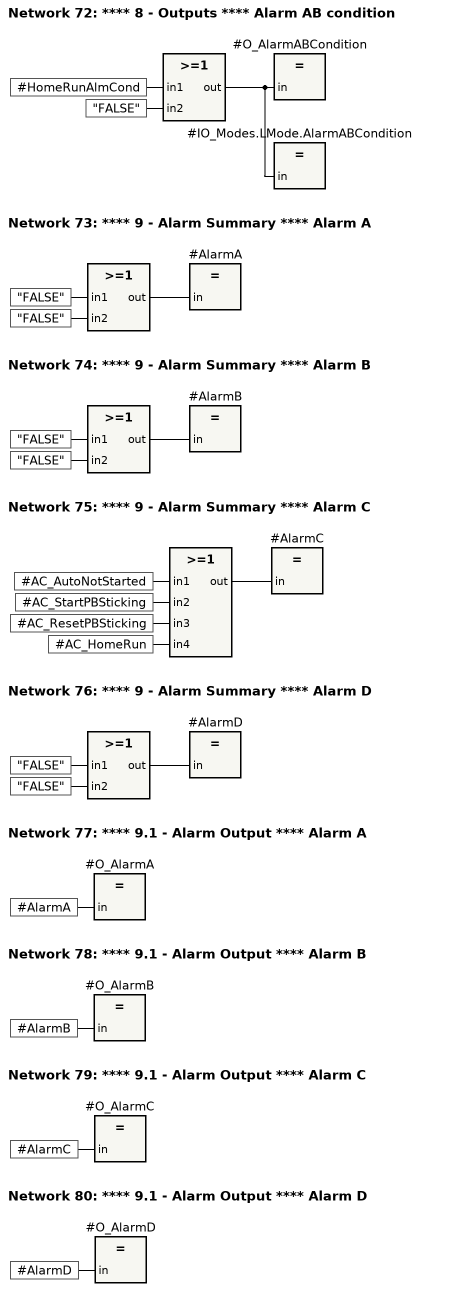
   #O_AlarmABCondition := #HomeRunAlmCond OR "FALSE";
   #IO_Modes.LMode.AlarmABCondition := #O_AlarmABCondition;
END_REGION

REGION Network 73: **** 9 - Alarm Summary **** Alarm A
   // Summary of alarms A
   #AlarmA := "FALSE" OR "FALSE";
END_REGION

REGION Network 74: **** 9 - Alarm Summary **** Alarm B
   // Summary of alarms B
   #AlarmB := "FALSE" OR "FALSE";
END_REGION

REGION Network 75: **** 9 - Alarm Summary **** Alarm C
   // Summary of alarms C
   #AlarmC := #AC_AutoNotStarted OR #AC_StartPBSticking OR #AC_ResetPBSticking OR #AC_HomeRun;
END_REGION

REGION Network 76: **** 9 - Alarm Summary **** Alarm D
   // Summary of alarms D
   #AlarmD := "FALSE" OR "FALSE";
END_REGION

REGION Network 77: **** 9.1 - Alarm Output **** Alarm A
   // Summary of alarms A
   #O_AlarmA := #AlarmA;
END_REGION

REGION Network 78: **** 9.1 - Alarm Output **** Alarm B
   // Summary of alarms B
   #O_AlarmB := #AlarmB;
END_REGION

REGION Network 79: **** 9.1 - Alarm Output **** Alarm C
   // Summary of alarms C
   #O_AlarmC := #AlarmC;
END_REGION

REGION Network 80: **** 9.1 - Alarm Output **** Alarm D
   // Summary of alarms D
   #O_AlarmD := #AlarmD;
END_REGION

REGION Network 81: **** 9.2 - Alarm DWord**** Alarm To DWord
   // Alarm Word
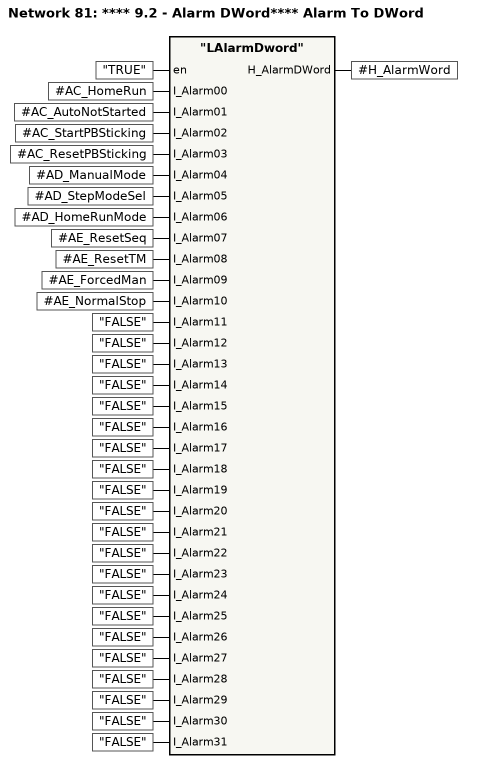
   IF "TRUE" THEN
       "LAlarmDword"(I_Alarm00 := #AC_HomeRun,
                     I_Alarm01 := #AC_AutoNotStarted,
                     I_Alarm02 := #AC_StartPBSticking,
                     I_Alarm03 := #AC_ResetPBSticking,
                     I_Alarm04 := #AD_ManualMode,
                     I_Alarm05 := #AD_StepModeSel,
                     I_Alarm06 := #AD_HomeRunMode,
                     I_Alarm07 := #AE_ResetSeq,
                     I_Alarm08 := #AE_ResetTM,
                     I_Alarm09 := #AE_ForcedMan,
                     I_Alarm10 := #AE_NormalStop,
                     I_Alarm11 := "FALSE",
                     I_Alarm12 := "FALSE",
                     I_Alarm13 := "FALSE",
                     I_Alarm14 := "FALSE",
                     I_Alarm15 := "FALSE",
                     I_Alarm16 := "FALSE",
                     I_Alarm17 := "FALSE",
                     I_Alarm18 := "FALSE",
                     I_Alarm19 := "FALSE",
                     I_Alarm20 := "FALSE",
                     I_Alarm21 := "FALSE",
                     I_Alarm22 := "FALSE",
                     I_Alarm23 := "FALSE",
                     I_Alarm24 := "FALSE",
                     I_Alarm25 := "FALSE",
                     I_Alarm26 := "FALSE",
                     I_Alarm27 := "FALSE",
                     I_Alarm28 := "FALSE",
                     I_Alarm29 := "FALSE",
                     I_Alarm30 := "FALSE",
                     I_Alarm31 := "FALSE",
                     H_AlarmDWord => #H_AlarmWord);
   END_IF;
END_REGION
END_FUNCTION_BLOCK

FUNCTION_BLOCK "LGeneralFunc"   // FB1001, FBD
TITLE = LGeneralFunc
{ S7_Optimized_Access := 'FALSE' }
AUTHOR : VCC
FAMILY : Control
NAME : GenFunc
VERSION : 1.0
// ================================================================================
// This module handles General Reverse Switch, General High Speed and Lamptest.
// It will also give the user and 8 bit interface for project specific functions.
// ================================================================================
// stored: AutoNumber false, IsIECCheckEnabled false, SetENOAutomatically False, UDAEnableTagReadback false
   VAR_INPUT
      I_GenRevSw { ExternalAccessible := 'False'; ExternalVisible := 'False'; ExternalWritable := 'False'} : Bool;   // General reverse switch
      I_GenHighSpeed { ExternalAccessible := 'False'; ExternalVisible := 'False'; ExternalWritable := 'False'} : Bool;   // General high speed
      I_Lamptest { ExternalAccessible := 'False'; ExternalVisible := 'False'; ExternalWritable := 'False'} : Bool;   // Lamptest PB
      I_LamptestSec { ExternalAccessible := 'False'; ExternalVisible := 'False'; ExternalWritable := 'False'} : Int := 60;   // The number of seconds that Lamptest will be on (Sec)
   END_VAR
   VAR_OUTPUT
      O_GeneralFunc : Word;   // General functions
      O_Lamptest { ExternalAccessible := 'False'; ExternalVisible := 'False'; ExternalWritable := 'False'} : Bool;   // Lamptest
      O_LamptestSteady { ExternalAccessible := 'False'; ExternalVisible := 'False'; ExternalWritable := 'False'} : Bool;   // Lamptest always on
      O_LamptestPBHMI { ExternalAccessible := 'False'; ExternalVisible := 'False'; ExternalWritable := 'False'} : Bool;   // Lamptest pushbutton HMI / Lamptest
      O_GenHighSpeed { ExternalAccessible := 'False'; ExternalVisible := 'False'; ExternalWritable := 'False'} : Bool;   // General High Speed
   END_VAR
   VAR_IN_OUT
      IO_Modes : "Modes";
   END_VAR
   VAR DB_SPECIFIC
      H_HMIGenFuncCmd : Word;   // General function commands from HMI
      AutoMode { ExternalAccessible := 'False'; ExternalVisible := 'False'; ExternalWritable := 'False'} : Bool;   // Auto mode
      AutoSel { ExternalAccessible := 'False'; ExternalVisible := 'False'; ExternalWritable := 'False'} : Bool;   // Auto is selected
      AlarmAB { ExternalAccessible := 'False'; ExternalVisible := 'False'; ExternalWritable := 'False'} : Bool;   // Alarm A or B is active
      HMIGenHighSpeed { ExternalAccessible := 'False'; ExternalVisible := 'False'; ExternalWritable := 'False'} : Bool;   // General High Speed for manual movement
      HMILamptest { ExternalAccessible := 'False'; ExternalVisible := 'False'; ExternalWritable := 'False'} : Bool;   // Lamptest
      GenHighSpeedSelected { ExternalAccessible := 'False'; ExternalVisible := 'False'; ExternalWritable := 'False'} : Bool;   // General high speed is selected
      LamptestSelected : Bool;   // Lamptest is selected
      PulseLamptest { ExternalAccessible := 'False'; ExternalVisible := 'False'; ExternalWritable := 'False'} : Bool;   // Pulse for lamptest
      PulseGenHighSpeed { ExternalAccessible := 'False'; ExternalVisible := 'False'; ExternalWritable := 'False'} : Bool;   // Pulse General high speed
      TimerLamptest { ExternalAccessible := 'False'; ExternalVisible := 'False'; ExternalWritable := 'False'} : Bool;   // Timer for Lamptest
      LamptestSec { ExternalAccessible := 'False'; ExternalVisible := 'False'; ExternalWritable := 'False'} : DInt;   // Lamptest on for xxx milliesec
      LamptestMillieSec { ExternalAccessible := 'False'; ExternalVisible := 'False'; ExternalWritable := 'False'} : DInt;   // Converted value
   END_VAR
   VAR
      TimerLampTestSel { ExternalAccessible := 'False'; ExternalVisible := 'False'; ExternalWritable := 'False'; S7_SetPoint := 'True'} : "LTimer";
   END_VAR
   VAR_TEMP
      SetLamptest : Bool;   // Set Lamptest
      ResetLamptest : Bool;   // Reset Lamptest
      ElapseTime : DInt;   // Elapse time for Lamptest
   END_VAR
   VAR_TEMP   // added for the SCL form of the ladder/FBD networks
      _w1 : Bool;
      _w2 : Bool;
   END_VAR
BEGIN

REGION Network 1: **** 1 - Inputs **** Extract the general functions from HMI
   // Extract the general functions from HMI
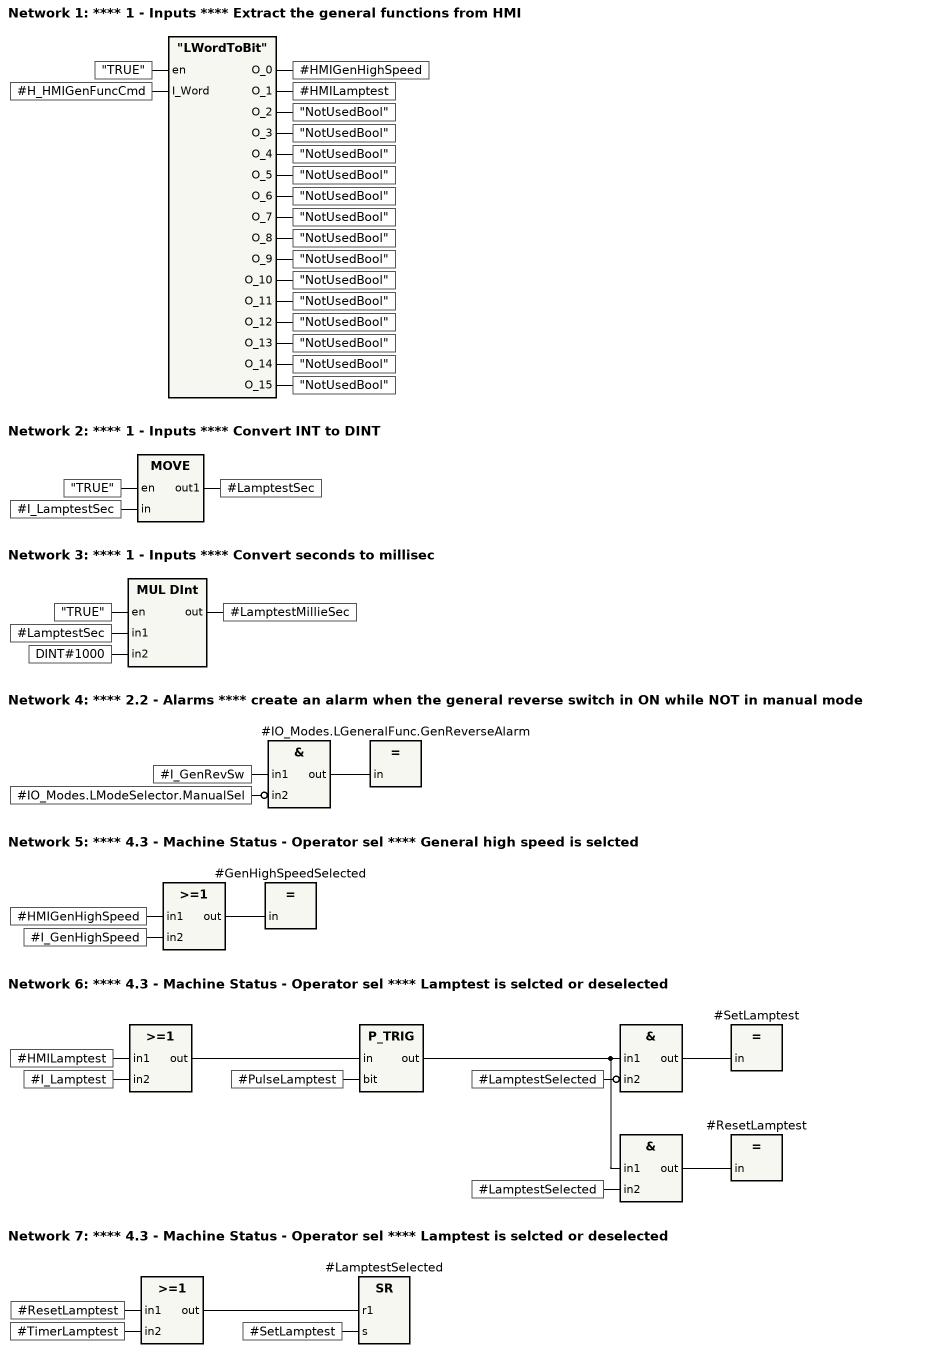
   IF "TRUE" THEN
       "LWordToBit"(I_Word := #H_HMIGenFuncCmd,
                    O_0 => #HMIGenHighSpeed,
                    O_1 => #HMILamptest,
                    O_2 => "NotUsedBool",
                    O_3 => "NotUsedBool",
                    O_4 => "NotUsedBool",
                    O_5 => "NotUsedBool",
                    O_6 => "NotUsedBool",
                    O_7 => "NotUsedBool",
                    O_8 => "NotUsedBool",
                    O_9 => "NotUsedBool",
                    O_10 => "NotUsedBool",
                    O_11 => "NotUsedBool",
                    O_12 => "NotUsedBool",
                    O_13 => "NotUsedBool",
                    O_14 => "NotUsedBool",
                    O_15 => "NotUsedBool");
   END_IF;
END_REGION

REGION Network 2: **** 1 - Inputs **** Convert INT to DINT
   // Convert INT to DINT
   IF "TRUE" THEN #LamptestSec := #I_LamptestSec; END_IF;
END_REGION

REGION Network 3: **** 1 - Inputs **** Convert seconds to millisec
   // Convert seconds to millisec
   IF "TRUE" THEN #LamptestMillieSec := #LamptestSec * DINT#1000; END_IF;
END_REGION

REGION Network 4: **** 2.2 - Alarms **** create an alarm when the general reverse switch in ON while NOT in manual mode
   // create an alarm when the general reverse switch in ON while NOT in manual mode
   #IO_Modes.LGeneralFunc.GenReverseAlarm := #I_GenRevSw AND NOT #IO_Modes.LModeSelector.ManualSel;
END_REGION

REGION Network 5: **** 4.3 - Machine Status - Operator sel **** General high speed is selcted
   // General high speed is selcted
   #GenHighSpeedSelected := #HMIGenHighSpeed OR #I_GenHighSpeed;
END_REGION

REGION Network 6: **** 4.3 - Machine Status - Operator sel **** Lamptest is selcted or deselected
   // Lamptest is selcted or deselected
   #_w1 := #HMILamptest OR #I_Lamptest;
   #_w2 := #_w1 AND NOT #PulseLamptest;   // rising edge
   #PulseLamptest := #_w1;
   #SetLamptest := #_w2 AND NOT #LamptestSelected;
   #ResetLamptest := #_w2 AND #LamptestSelected;
END_REGION

REGION Network 7: **** 4.3 - Machine Status - Operator sel **** Lamptest is selcted or deselected
   // Lamptest is selcted or deselected
   IF #SetLamptest THEN
       #LamptestSelected := TRUE;   // SR flip-flop
   END_IF;
   IF #ResetLamptest OR #TimerLamptest THEN #LamptestSelected := FALSE; END_IF;
END_REGION

REGION Network 8: **** 4.3 - Machine Status - Operator sel **** Timer for Lamptest
   // Timer for Lamptest
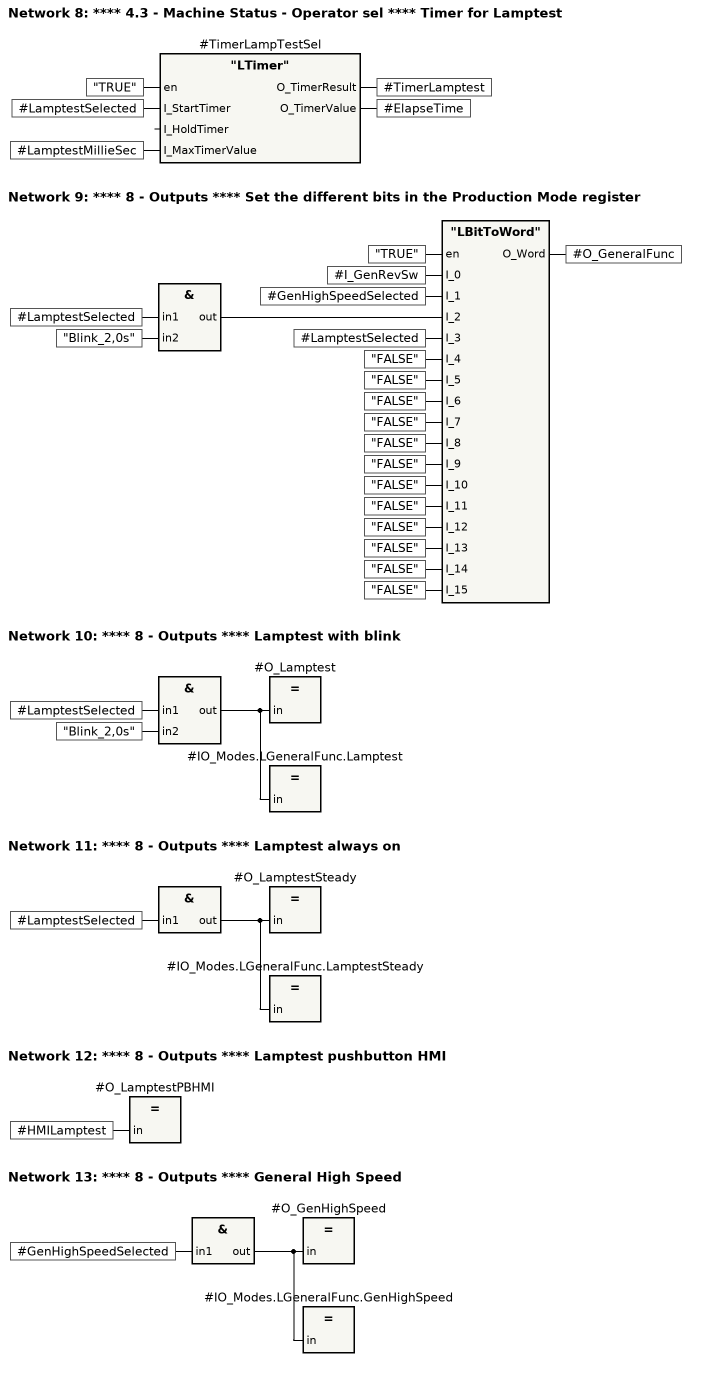
   IF "TRUE" THEN
       #TimerLampTestSel(I_StartTimer := #LamptestSelected,   // "LTimer"
                         I_MaxTimerValue := #LamptestMillieSec,
                         O_TimerResult => #TimerLamptest,
                         O_TimerValue => #ElapseTime);
   END_IF;
END_REGION

REGION Network 9: **** 8 - Outputs **** Set the different bits in the Production Mode register
   // Set the different bits in the Production Mode register
   IF "TRUE" THEN
       "LBitToWord"(I_0 := #I_GenRevSw,
                    I_1 := #GenHighSpeedSelected,
                    I_2 := #LamptestSelected AND "Blink_2,0s",
                    I_3 := #LamptestSelected,
                    I_4 := "FALSE",
                    I_5 := "FALSE",
                    I_6 := "FALSE",
                    I_7 := "FALSE",
                    I_8 := "FALSE",
                    I_9 := "FALSE",
                    I_10 := "FALSE",
                    I_11 := "FALSE",
                    I_12 := "FALSE",
                    I_13 := "FALSE",
                    I_14 := "FALSE",
                    I_15 := "FALSE",
                    O_Word => #O_GeneralFunc);
   END_IF;
END_REGION

REGION Network 10: **** 8 - Outputs **** Lamptest with blink
   // Lamptest with blink
   #O_Lamptest := #LamptestSelected AND "Blink_2,0s";
   #IO_Modes.LGeneralFunc.Lamptest := #O_Lamptest;
END_REGION

REGION Network 11: **** 8 - Outputs **** Lamptest always on
   // Lamptest always on
   #O_LamptestSteady := #LamptestSelected;
   #IO_Modes.LGeneralFunc.LamptestSteady := #LamptestSelected;
END_REGION

REGION Network 12: **** 8 - Outputs **** Lamptest pushbutton HMI
   #O_LamptestPBHMI := #HMILamptest;
END_REGION

REGION Network 13: **** 8 - Outputs **** General High Speed
   // General High Speed
   #O_GenHighSpeed := #GenHighSpeedSelected;
   #IO_Modes.LGeneralFunc.GenHighSpeed := #GenHighSpeedSelected;
END_REGION

REGION Network 14: **** 8 - Outputs **** General Reverse Switch
   // General Reverse Switch
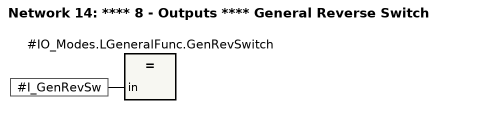
   #IO_Modes.LGeneralFunc.GenRevSwitch := #I_GenRevSw;
END_REGION
END_FUNCTION_BLOCK

FUNCTION_BLOCK "LModeSelector"   // FB1002, FBD
TITLE = LModeSelector
{ S7_Optimized_Access := 'FALSE' }
AUTHOR : VCC
FAMILY : Control
NAME : ModeSel
VERSION : 1.0
// ================================================================================
// This module handles that only one mode is selected in the modezon, it also 
// handle interlocking between the HMIs. Each modezone can have 5 HMI.
// ================================================================================
// stored: AutoNumber false, IsIECCheckEnabled false, SetENOAutomatically False, UDAEnableTagReadback false
   VAR_INPUT
      I_NumHMI { ExternalAccessible := 'False'; ExternalVisible := 'False'; ExternalWritable := 'False'} : Int;   // Number of HMI used in the modezon
      I_LockManualTime { ExternalAccessible := 'False'; ExternalVisible := 'False'; ExternalWritable := 'False'} : Int;   // The number of seconds that Lock Manual shall be active
      I_StartPB { ExternalAccessible := 'False'; ExternalVisible := 'False'; ExternalWritable := 'False'} : Bool;   // Summary of Start buttons
      I_AlarmResetPB { ExternalAccessible := 'False'; ExternalVisible := 'False'; ExternalWritable := 'False'} : Bool;   // Summary of Alarm reset buttons
      I_SafetyNotOk { ExternalAccessible := 'False'; ExternalVisible := 'False'; ExternalWritable := 'False'} : Bool;   // Safety is not ok
      I_FailSafeResetAck { ExternalAccessible := 'False'; ExternalVisible := 'False'; ExternalWritable := 'False'} : Bool;   // F_Ack_Op FB in safety program is requesting value 9 on FailSafeReset output
      I_FailSafeAckID { ExternalAccessible := 'False'; ExternalVisible := 'False'; ExternalWritable := 'False'} : Int;   // F_Ack ID
      I_AllHMIAutoSel { ExternalAccessible := 'False'; ExternalVisible := 'False'; ExternalWritable := 'False'} : Bool;   // All HMI to Auto Selected
      I_HMI1ForceMan { ExternalAccessible := 'False'; ExternalVisible := 'False'; ExternalWritable := 'False'} : Bool;   // Forced manual selected on HMI1
      I_HMI1SetPB { ExternalAccessible := 'False'; ExternalVisible := 'False'; ExternalWritable := 'False'} : Bool;   // Set PB activated on HMI1
      I_HMI1ResetPB { ExternalAccessible := 'False'; ExternalVisible := 'False'; ExternalWritable := 'False'} : Bool;   // Reset PB activated on HMI1
      I_HMI1StartPB { ExternalAccessible := 'False'; ExternalVisible := 'False'; ExternalWritable := 'False'} : Bool;   // Start PB activated on HMI1
      I_HMI1AlarmResetPB { ExternalAccessible := 'False'; ExternalVisible := 'False'; ExternalWritable := 'False'} : Bool;   // AlarmReset PB activated on HMI1
      I_HMI2ForceMan { ExternalAccessible := 'False'; ExternalVisible := 'False'; ExternalWritable := 'False'} : Bool;   // Forced manual selected on HMI2
      I_HMI2SetPB { ExternalAccessible := 'False'; ExternalVisible := 'False'; ExternalWritable := 'False'} : Bool;   // Set PB activated on HMI2
      I_HMI2ResetPB { ExternalAccessible := 'False'; ExternalVisible := 'False'; ExternalWritable := 'False'} : Bool;   // Reset PB activated on HMI2
      I_HMI2StartPB { ExternalAccessible := 'False'; ExternalVisible := 'False'; ExternalWritable := 'False'} : Bool;   // Start PB activated on HMI2
      I_HMI2AlarmResetPB { ExternalAccessible := 'False'; ExternalVisible := 'False'; ExternalWritable := 'False'} : Bool;   // AlarmReset PB activated on HMI2
      I_HMI3ForceMan { ExternalAccessible := 'False'; ExternalVisible := 'False'; ExternalWritable := 'False'} : Bool;   // Forced manual selected on HMI3
      I_HMI3SetPB { ExternalAccessible := 'False'; ExternalVisible := 'False'; ExternalWritable := 'False'} : Bool;   // Set PB activated on HMI3
      I_HMI3ResetPB { ExternalAccessible := 'False'; ExternalVisible := 'False'; ExternalWritable := 'False'} : Bool;   // Reset PB activated on HMI3
      I_HMI3StartPB { ExternalAccessible := 'False'; ExternalVisible := 'False'; ExternalWritable := 'False'} : Bool;   // Start PB activated on HMI
      I_HMI3AlarmResetPB { ExternalAccessible := 'False'; ExternalVisible := 'False'; ExternalWritable := 'False'} : Bool;   // AlarmReset PB activated on HMI3
      I_HMI4ForceMan { ExternalAccessible := 'False'; ExternalVisible := 'False'; ExternalWritable := 'False'} : Bool;   // Forced manual selected on HMI4
      I_HMI4SetPB { ExternalAccessible := 'False'; ExternalVisible := 'False'; ExternalWritable := 'False'} : Bool;   // Set PB activated on HMI4
      I_HMI4ResetPB { ExternalAccessible := 'False'; ExternalVisible := 'False'; ExternalWritable := 'False'} : Bool;   // Reset PB activated on HMI4
      I_HMI4StartPB { ExternalAccessible := 'False'; ExternalVisible := 'False'; ExternalWritable := 'False'} : Bool;   // Start PB activated on HMI4
      I_HMI4AlarmResetPB { ExternalAccessible := 'False'; ExternalVisible := 'False'; ExternalWritable := 'False'} : Bool;   // AlarmReset PB activated on HMI4
      I_HMI5ForceMan { ExternalAccessible := 'False'; ExternalVisible := 'False'; ExternalWritable := 'False'} : Bool;   // Forced manual selected on HMI5
      I_HMI5SetPB { ExternalAccessible := 'False'; ExternalVisible := 'False'; ExternalWritable := 'False'} : Bool;   // Set PB activated on HMI5
      I_HMI5ResetPB { ExternalAccessible := 'False'; ExternalVisible := 'False'; ExternalWritable := 'False'} : Bool;   // Reset PB activated on HMI5
      I_HMI5StartPB { ExternalAccessible := 'False'; ExternalVisible := 'False'; ExternalWritable := 'False'} : Bool;   // Start PB activated on HMI5
      I_HMI5AlarmResetPB { ExternalAccessible := 'False'; ExternalVisible := 'False'; ExternalWritable := 'False'} : Bool;   // AlarmReset PB activated on HMI5
   END_VAR
   VAR_OUTPUT
      O_AutoSel { ExternalAccessible := 'False'; ExternalVisible := 'False'; ExternalWritable := 'False'} : Bool;   // Auto selected
      O_AllAutoSel { ExternalAccessible := 'False'; ExternalVisible := 'False'; ExternalWritable := 'False'} : Bool;   // All objects in Auto selected
      O_StepSel { ExternalAccessible := 'False'; ExternalVisible := 'False'; ExternalWritable := 'False'} : Bool;   // Step selected
      O_HomeRunSel { ExternalAccessible := 'False'; ExternalVisible := 'False'; ExternalWritable := 'False'} : Bool;   // Homerun selected
      O_ManualSel { ExternalAccessible := 'False'; ExternalVisible := 'False'; ExternalWritable := 'False'} : Bool;   // Manual selected
      O_ForcedManActSel { ExternalAccessible := 'False'; ExternalVisible := 'False'; ExternalWritable := 'False'} : Bool;   // Forced manual selected
      O_PBSetSel { ExternalAccessible := 'False'; ExternalVisible := 'False'; ExternalWritable := 'False'} : Bool;   // Set selected
      O_PBResetSel { ExternalAccessible := 'False'; ExternalVisible := 'False'; ExternalWritable := 'False'} : Bool;   // Reset selected
      O_StartPBSel { ExternalAccessible := 'False'; ExternalVisible := 'False'; ExternalWritable := 'False'} : Bool;   // Start is activated
      O_AlarmResetPBSel { ExternalAccessible := 'False'; ExternalVisible := 'False'; ExternalWritable := 'False'} : Bool;   // Alarm reset is activated
      O_ResetTMSel { ExternalAccessible := 'False'; ExternalVisible := 'False'; ExternalWritable := 'False'} : Bool;   // Reset transport memory
      O_ResetSeqSel { ExternalAccessible := 'False'; ExternalVisible := 'False'; ExternalWritable := 'False'} : Bool;   // Reset squence
      O_CycleFinishedSel { ExternalAccessible := 'False'; ExternalVisible := 'False'; ExternalWritable := 'False'} : Bool;   // Cycle finished selected
      O_HomeRunRedoSel { ExternalAccessible := 'False'; ExternalVisible := 'False'; ExternalWritable := 'False'} : Bool;   // Redo after Homerun selected
      O_HomeRunWorkDoneSel { ExternalAccessible := 'False'; ExternalVisible := 'False'; ExternalWritable := 'False'} : Bool;   // WorkDone after Homerun selected
   END_VAR
   VAR_IN_OUT
      IO_FailsafeReset { ExternalAccessible := 'False'; ExternalVisible := 'False'; ExternalWritable := 'False'} : Int;   // Number to Failsafe to reset safety
   END_VAR
   VAR DB_SPECIFIC
      H_HMIHomeRunModeCmd : Word;   // Homerun Mode commands from HMI
      H_Anim : Word;   // Animation for HMI
      H_ActiveHMI : Int;   // Active HMI
      H_NameActiveHMI : String[25];   // Name of the Active HMI
      H_LockManTime : Int;   // Lock manual time
      H_HMI1ModeCmd : Word;   // Mode commands from HMI1
      H_HMI2ModeCmd : Word;   // Mode commands from HMI2
      H_HMI3ModeCmd : Word;   // Mode commands from HMI3
      H_HMI4ModeCmd : Word;   // Mode commands from HMI4
      H_HMI5ModeCmd : Word;   // Mode commands from HMI5. For operator panels, no S7_m_c
      HMI1AutoSel { ExternalAccessible := 'False'; ExternalVisible := 'False'; ExternalWritable := 'False'} : Bool;   // Auto selected on HMI1
      HMI1StepSel { ExternalAccessible := 'False'; ExternalVisible := 'False'; ExternalWritable := 'False'} : Bool;   // Step selected on HMI1
      HMI1HomeRunSel { ExternalAccessible := 'False'; ExternalVisible := 'False'; ExternalWritable := 'False'} : Bool;   // Homerun selected on HMI1
      HMI1ManualSel { ExternalAccessible := 'False'; ExternalVisible := 'False'; ExternalWritable := 'False'} : Bool;   // Manual selected on HMI1
      HMI1LockManual { ExternalAccessible := 'False'; ExternalVisible := 'False'; ExternalWritable := 'False'} : Bool;   // Lock manual for HMI1
      HMI1AllHMIAutoSel { ExternalAccessible := 'False'; ExternalVisible := 'False'; ExternalWritable := 'False'} : Bool;   // All HMI Auto selected on HMI1
      HMI1Start { ExternalAccessible := 'False'; ExternalVisible := 'False'; ExternalWritable := 'False'} : Bool;   // Start on HMI1
      HMI1AlarmReset { ExternalAccessible := 'False'; ExternalVisible := 'False'; ExternalWritable := 'False'} : Bool;   // AlarmReset on HMI1
      HMI1ResetTM { ExternalAccessible := 'False'; ExternalVisible := 'False'; ExternalWritable := 'False'} : Bool;   // Reset transport memory from HMI1
      HMI1ResetSeq { ExternalAccessible := 'False'; ExternalVisible := 'False'; ExternalWritable := 'False'} : Bool;   // Reset sequence from HMI1
      HMI1CycleFinished { ExternalAccessible := 'False'; ExternalVisible := 'False'; ExternalWritable := 'False'} : Bool;   // Cycle Finished from HMI1
      HMI1AlarmResetAck { ExternalAccessible := 'False'; ExternalVisible := 'False'; ExternalWritable := 'False'} : Bool;   // Alarm Reset acknowledge from HMI1
      HMI2AutoSel { ExternalAccessible := 'False'; ExternalVisible := 'False'; ExternalWritable := 'False'} : Bool;   // Auto selected on HMI2
      HMI2StepSel { ExternalAccessible := 'False'; ExternalVisible := 'False'; ExternalWritable := 'False'} : Bool;   // Step selected on HMI2
      HMI2HomeRunSel { ExternalAccessible := 'False'; ExternalVisible := 'False'; ExternalWritable := 'False'} : Bool;   // Homerun selected on HMI2
      HMI2ManualSel { ExternalAccessible := 'False'; ExternalVisible := 'False'; ExternalWritable := 'False'} : Bool;   // Manual selected on HMI2
      HMI2LockManual { ExternalAccessible := 'False'; ExternalVisible := 'False'; ExternalWritable := 'False'} : Bool;   // Lock manual for HMI2
      HMI2AllHMIAutoSel { ExternalAccessible := 'False'; ExternalVisible := 'False'; ExternalWritable := 'False'} : Bool;   // All HMI Auto selected on HMI2
      HMI2Start { ExternalAccessible := 'False'; ExternalVisible := 'False'; ExternalWritable := 'False'} : Bool;   // Start on HMI2
      HMI2AlarmReset { ExternalAccessible := 'False'; ExternalVisible := 'False'; ExternalWritable := 'False'} : Bool;   // AlarmReset on HMI2
      HMI2ResetTM { ExternalAccessible := 'False'; ExternalVisible := 'False'; ExternalWritable := 'False'} : Bool;   // Reset transport memory from HMI2
      HMI2ResetSeq { ExternalAccessible := 'False'; ExternalVisible := 'False'; ExternalWritable := 'False'} : Bool;   // Reset sequence from HMI2
      HMI2CycleFinished { ExternalAccessible := 'False'; ExternalVisible := 'False'; ExternalWritable := 'False'} : Bool;   // Cycle Finished from HMI2
      HMI2AlarmResetAck { ExternalAccessible := 'False'; ExternalVisible := 'False'; ExternalWritable := 'False'} : Bool;   // Alarm Reset acknowledge from HMI2
      HMI3AutoSel { ExternalAccessible := 'False'; ExternalVisible := 'False'; ExternalWritable := 'False'} : Bool;   // Auto selected on HMI3
      HMI3StepSel { ExternalAccessible := 'False'; ExternalVisible := 'False'; ExternalWritable := 'False'} : Bool;   // Step selected on HMI3
      HMI3HomeRunSel { ExternalAccessible := 'False'; ExternalVisible := 'False'; ExternalWritable := 'False'} : Bool;   // Homerun selected on HMI3
      HMI3ManualSel { ExternalAccessible := 'False'; ExternalVisible := 'False'; ExternalWritable := 'False'} : Bool;   // Manual selected on HMI3
      HMI3LockManual { ExternalAccessible := 'False'; ExternalVisible := 'False'; ExternalWritable := 'False'} : Bool;   // Lock manual for HMI3
      HMI3AllHMIAutoSel { ExternalAccessible := 'False'; ExternalVisible := 'False'; ExternalWritable := 'False'} : Bool;   // All HMI Auto selected on HMI3
      HMI3Start { ExternalAccessible := 'False'; ExternalVisible := 'False'; ExternalWritable := 'False'} : Bool;   // Start on HMI3
      HMI3AlarmReset { ExternalAccessible := 'False'; ExternalVisible := 'False'; ExternalWritable := 'False'} : Bool;   // AlarmReset on HMI3
      HMI3ResetTM { ExternalAccessible := 'False'; ExternalVisible := 'False'; ExternalWritable := 'False'} : Bool;   // Reset transport memory from HMI3
      HMI3ResetSeq { ExternalAccessible := 'False'; ExternalVisible := 'False'; ExternalWritable := 'False'} : Bool;   // Reset sequence from HMI3
      HMI3CycleFinished { ExternalAccessible := 'False'; ExternalVisible := 'False'; ExternalWritable := 'False'} : Bool;   // Cycle Finished from HMI3
      HMI3AlarmResetAck { ExternalAccessible := 'False'; ExternalVisible := 'False'; ExternalWritable := 'False'} : Bool;   // Alarm Reset acknowledge from 3
      HMI4AutoSel { ExternalAccessible := 'False'; ExternalVisible := 'False'; ExternalWritable := 'False'} : Bool;   // Auto selected on HMI4
      HMI4StepSel { ExternalAccessible := 'False'; ExternalVisible := 'False'; ExternalWritable := 'False'} : Bool;   // Step selected on HMI4
      HMI4HomeRunSel { ExternalAccessible := 'False'; ExternalVisible := 'False'; ExternalWritable := 'False'} : Bool;   // Homerun selected on HMI4
      HMI4ManualSel { ExternalAccessible := 'False'; ExternalVisible := 'False'; ExternalWritable := 'False'} : Bool;   // Manual selected on HMI4
      HMI4LockManual { ExternalAccessible := 'False'; ExternalVisible := 'False'; ExternalWritable := 'False'} : Bool;   // Lock manual for HMI4
      HMI4AllHMIAutoSel { ExternalAccessible := 'False'; ExternalVisible := 'False'; ExternalWritable := 'False'} : Bool;   // All HMI Auto selected on HMI4
      HMI4Start { ExternalAccessible := 'False'; ExternalVisible := 'False'; ExternalWritable := 'False'} : Bool;   // Start on HMI4
      HMI4AlarmReset { ExternalAccessible := 'False'; ExternalVisible := 'False'; ExternalWritable := 'False'} : Bool;   // AlarmReset on HMI4
      HMI4ResetTM { ExternalAccessible := 'False'; ExternalVisible := 'False'; ExternalWritable := 'False'} : Bool;   // Reset transport memory from HMI4
      HMI4ResetSeq { ExternalAccessible := 'False'; ExternalVisible := 'False'; ExternalWritable := 'False'} : Bool;   // Reset sequence from HMI4
      HMI4CycleFinished { ExternalAccessible := 'False'; ExternalVisible := 'False'; ExternalWritable := 'False'} : Bool;   // Cycle Finished from HMI4
      HMI4AlarmResetAck { ExternalAccessible := 'False'; ExternalVisible := 'False'; ExternalWritable := 'False'} : Bool;   // Alarm Reset acknowledge from HMI4
      HMI5AutoSel { ExternalAccessible := 'False'; ExternalVisible := 'False'; ExternalWritable := 'False'} : Bool;   // Auto selected on HMI5
      HMI5StepSel { ExternalAccessible := 'False'; ExternalVisible := 'False'; ExternalWritable := 'False'} : Bool;   // Step selected on HMI5
      HMI5HomeRunSel { ExternalAccessible := 'False'; ExternalVisible := 'False'; ExternalWritable := 'False'} : Bool;   // Homerun selected on HMI5
      HMI5ManualSel { ExternalAccessible := 'False'; ExternalVisible := 'False'; ExternalWritable := 'False'} : Bool;   // Manual selected on HMI5
      HMI5LockManual { ExternalAccessible := 'False'; ExternalVisible := 'False'; ExternalWritable := 'False'} : Bool;   // Lock manual for HMI5
      HMI5AllHMIAutoSel { ExternalAccessible := 'False'; ExternalVisible := 'False'; ExternalWritable := 'False'} : Bool;   // All HMI Auto selected on HMI5
      HMI5Start { ExternalAccessible := 'False'; ExternalVisible := 'False'; ExternalWritable := 'False'} : Bool;   // Start on HMI5
      HMI5AlarmReset { ExternalAccessible := 'False'; ExternalVisible := 'False'; ExternalWritable := 'False'} : Bool;   // AlarmReset on HMI5
      HMI5ResetTM { ExternalAccessible := 'False'; ExternalVisible := 'False'; ExternalWritable := 'False'} : Bool;   // Reset transport memory from HMI5
      HMI5ResetSeq { ExternalAccessible := 'False'; ExternalVisible := 'False'; ExternalWritable := 'False'} : Bool;   // Reset sequence from HMI5
      HMI5CycleFinished { ExternalAccessible := 'False'; ExternalVisible := 'False'; ExternalWritable := 'False'} : Bool;   // Cycle Finished from HMI5
      HMI5AlarmResetAck { ExternalAccessible := 'False'; ExternalVisible := 'False'; ExternalWritable := 'False'} : Bool;   // Alarm Reset acknowledge from HMI5
      HMIHomeRunRedo { ExternalAccessible := 'False'; ExternalVisible := 'False'; ExternalWritable := 'False'} : Bool;   // Redo after homerun from HMI
      HMIHomeRunWorkDone { ExternalAccessible := 'False'; ExternalVisible := 'False'; ExternalWritable := 'False'} : Bool;   // WorkDone after homerun from HMI
      LockManualTimeout { ExternalAccessible := 'False'; ExternalVisible := 'False'; ExternalWritable := 'False'} : Bool;   // Lock manual button timeout
      AllHmiAutoSel { ExternalAccessible := 'False'; ExternalVisible := 'False'; ExternalWritable := 'False'} : Bool;   // All Hmi Auto selected
      AlarmResetPBSel { ExternalAccessible := 'False'; ExternalVisible := 'False'; ExternalWritable := 'False'} : Bool;   // Alarm reset is activated
      AlarmResetPBSelReset { ExternalAccessible := 'False'; ExternalVisible := 'False'; ExternalWritable := 'False'} : Bool;   // Reset AlarmResetPBSel after predefined time
      AlarmResetPBSelResetPE { ExternalAccessible := 'False'; ExternalVisible := 'False'; ExternalWritable := 'False'} : Bool;   // Positive edge of AlarmResetPbSelReset
      FailSafeReset6Pulse { ExternalAccessible := 'False'; ExternalVisible := 'False'; ExternalWritable := 'False'} : Bool;   // Pulse to set value 6 on FailSafeReset Output
      FailSafeReset9Pulse { ExternalAccessible := 'False'; ExternalVisible := 'False'; ExternalWritable := 'False'} : Bool;   // Pulse to set value 9 on FailSafeReset Output
      ResetAlarmAckMemPulse { ExternalAccessible := 'False'; ExternalVisible := 'False'; ExternalWritable := 'False'} : Bool;   // Pulse to reset AlarmResetAckMem on negative edge of I_FailSafeResetAck
      AlarmResetAckMem { ExternalAccessible := 'False'; ExternalVisible := 'False'; ExternalWritable := 'False'} : Bool;   // memory : Pushbutton AlarmResetAck has been pushed on HMI
      StartPBSel { ExternalAccessible := 'False'; ExternalVisible := 'False'; ExternalWritable := 'False'} : Bool;   // Summary of the Start push buttons
      AutoSel { ExternalAccessible := 'False'; ExternalVisible := 'False'; ExternalWritable := 'False'} : Bool;   // Auto selected
      HMIStartPE { ExternalAccessible := 'False'; ExternalVisible := 'False'; ExternalWritable := 'False'} : Bool;   // Positive edge on start button from HMI
      HMIResetTMPE { ExternalAccessible := 'False'; ExternalVisible := 'False'; ExternalWritable := 'False'} : Bool;   // Positive edge on ResetTM button from HMI
      HMIResetSeqPE { ExternalAccessible := 'False'; ExternalVisible := 'False'; ExternalWritable := 'False'} : Bool;   // Positive edge on ResetSeq button from HMI
      HMIAlarmResetAckPE { ExternalAccessible := 'False'; ExternalVisible := 'False'; ExternalWritable := 'False'} : Bool;   // Positive edge on AlarmResetAck button from HMI
      HMILockManualPE { ExternalAccessible := 'False'; ExternalVisible := 'False'; ExternalWritable := 'False'} : Bool;   // Positive edge on LockManual button from HMI
      PBSetSel { ExternalAccessible := 'False'; ExternalVisible := 'False'; ExternalWritable := 'False'} : Bool;   // Set selected
      PBResetSel { ExternalAccessible := 'False'; ExternalVisible := 'False'; ExternalWritable := 'False'} : Bool;   // Reset selected
      CheckHMIActive { ExternalAccessible := 'False'; ExternalVisible := 'False'; ExternalWritable := 'False'} : Bool;   // Check Active HMI
      FailsafeReset { ExternalAccessible := 'False'; ExternalVisible := 'False'; ExternalWritable := 'False'} : Int;   // Number to Failsafe to reset safety
      ActiveHMI { ExternalAccessible := 'False'; ExternalVisible := 'False'; ExternalWritable := 'False'} : Int;   // Help memory for Active HMI
      LockManualSec { ExternalAccessible := 'False'; ExternalVisible := 'False'; ExternalWritable := 'False'} : DInt;   // Lock manual on for xxx milliesec
      LockManualMillieSec { ExternalAccessible := 'False'; ExternalVisible := 'False'; ExternalWritable := 'False'} : DInt;   // Converted value
      TimerLockManValue { ExternalAccessible := 'False'; ExternalVisible := 'False'; ExternalWritable := 'False'} : DInt;   // Timer value
   END_VAR
   VAR
      TimerLockMan { ExternalAccessible := 'False'; ExternalVisible := 'False'; ExternalWritable := 'False'; S7_SetPoint := 'True'} : "LTimer";   // Timer on Lock manual
      TimerAlarmResetPB { ExternalAccessible := 'False'; ExternalVisible := 'False'; ExternalWritable := 'False'; S7_SetPoint := 'True'} : "LTimer";   // Timer on alarm reset
   END_VAR
   VAR DB_SPECIFIC
      CheckActiveHMI { ExternalAccessible := 'False'; ExternalVisible := 'False'; ExternalWritable := 'False'; S7_SetPoint := 'True'} : TP_TIME;   // Timer
      CheckActiveHMI_1 { ExternalAccessible := 'False'; ExternalVisible := 'False'; ExternalWritable := 'False'; S7_SetPoint := 'True'} : TP_TIME;   // Timer
      CheckActiveHMI_2 { ExternalAccessible := 'False'; ExternalVisible := 'False'; ExternalWritable := 'False'; S7_SetPoint := 'True'} : TON_TIME;   // Timer
      CheckActiveHMI_3 { ExternalAccessible := 'False'; ExternalVisible := 'False'; ExternalWritable := 'False'; S7_SetPoint := 'True'} : TON_TIME;   // Timer
   END_VAR
   VAR_TEMP
      PHMI1AutoSel : Bool;   // Pulse Auto selected HMI1
      PHMI2AutoSel : Bool;   // Pulse Auto selected HMI2
      PHMI3AutoSel : Bool;   // Pulse Auto selected HMI3
      PHMI4AutoSel : Bool;   // Pulse Auto selected HMI4
      PHMI5AutoSel : Bool;   // Pulse Auto selected HMI5
      LockManualTime : Int;   // Lock manual time
      LockManualTimeInt : Int;   // Lock manual time
      LockManualTimeDInt : DInt;   // Lock manual time
   END_VAR
   VAR_TEMP   // added for the SCL form of the ladder/FBD networks
      _w1 : Bool;
      _w2 : Bool;
      _w3 : Bool;
      _w4 : Bool;
      _w5 : Bool;
   END_VAR
BEGIN

REGION Network 1: **** 1 - Inputs **** Extract the modeselection from HMI 1
   // Extract the modeselection from HMI 1
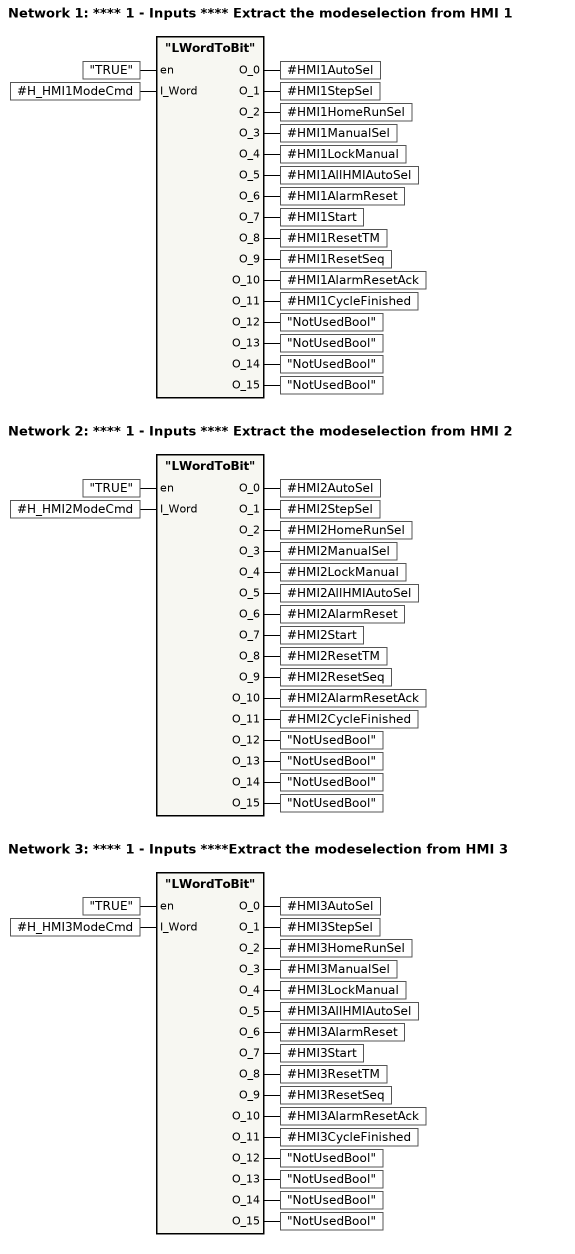
   IF "TRUE" THEN
       "LWordToBit"(I_Word := #H_HMI1ModeCmd,
                    O_0 => #HMI1AutoSel,
                    O_1 => #HMI1StepSel,
                    O_2 => #HMI1HomeRunSel,
                    O_3 => #HMI1ManualSel,
                    O_4 => #HMI1LockManual,
                    O_5 => #HMI1AllHMIAutoSel,
                    O_6 => #HMI1AlarmReset,
                    O_7 => #HMI1Start,
                    O_8 => #HMI1ResetTM,
                    O_9 => #HMI1ResetSeq,
                    O_10 => #HMI1AlarmResetAck,
                    O_11 => #HMI1CycleFinished,
                    O_12 => "NotUsedBool",
                    O_13 => "NotUsedBool",
                    O_14 => "NotUsedBool",
                    O_15 => "NotUsedBool");
   END_IF;
END_REGION

REGION Network 2: **** 1 - Inputs **** Extract the modeselection from HMI 2
   // Extract the modeselection from HMI 2
   IF "TRUE" THEN
       "LWordToBit"(I_Word := #H_HMI2ModeCmd,
                    O_0 => #HMI2AutoSel,
                    O_1 => #HMI2StepSel,
                    O_2 => #HMI2HomeRunSel,
                    O_3 => #HMI2ManualSel,
                    O_4 => #HMI2LockManual,
                    O_5 => #HMI2AllHMIAutoSel,
                    O_6 => #HMI2AlarmReset,
                    O_7 => #HMI2Start,
                    O_8 => #HMI2ResetTM,
                    O_9 => #HMI2ResetSeq,
                    O_10 => #HMI2AlarmResetAck,
                    O_11 => #HMI2CycleFinished,
                    O_12 => "NotUsedBool",
                    O_13 => "NotUsedBool",
                    O_14 => "NotUsedBool",
                    O_15 => "NotUsedBool");
   END_IF;
END_REGION

REGION Network 3: **** 1 - Inputs ****Extract the modeselection from HMI 3
   // Extract the modeselection from HMI 3
   IF "TRUE" THEN
       "LWordToBit"(I_Word := #H_HMI3ModeCmd,
                    O_0 => #HMI3AutoSel,
                    O_1 => #HMI3StepSel,
                    O_2 => #HMI3HomeRunSel,
                    O_3 => #HMI3ManualSel,
                    O_4 => #HMI3LockManual,
                    O_5 => #HMI3AllHMIAutoSel,
                    O_6 => #HMI3AlarmReset,
                    O_7 => #HMI3Start,
                    O_8 => #HMI3ResetTM,
                    O_9 => #HMI3ResetSeq,
                    O_10 => #HMI3AlarmResetAck,
                    O_11 => #HMI3CycleFinished,
                    O_12 => "NotUsedBool",
                    O_13 => "NotUsedBool",
                    O_14 => "NotUsedBool",
                    O_15 => "NotUsedBool");
   END_IF;
END_REGION

REGION Network 4: **** 1 - Inputs **** Extract the modeselection from HMI 4
   // Extract the modeselection from HMI 4
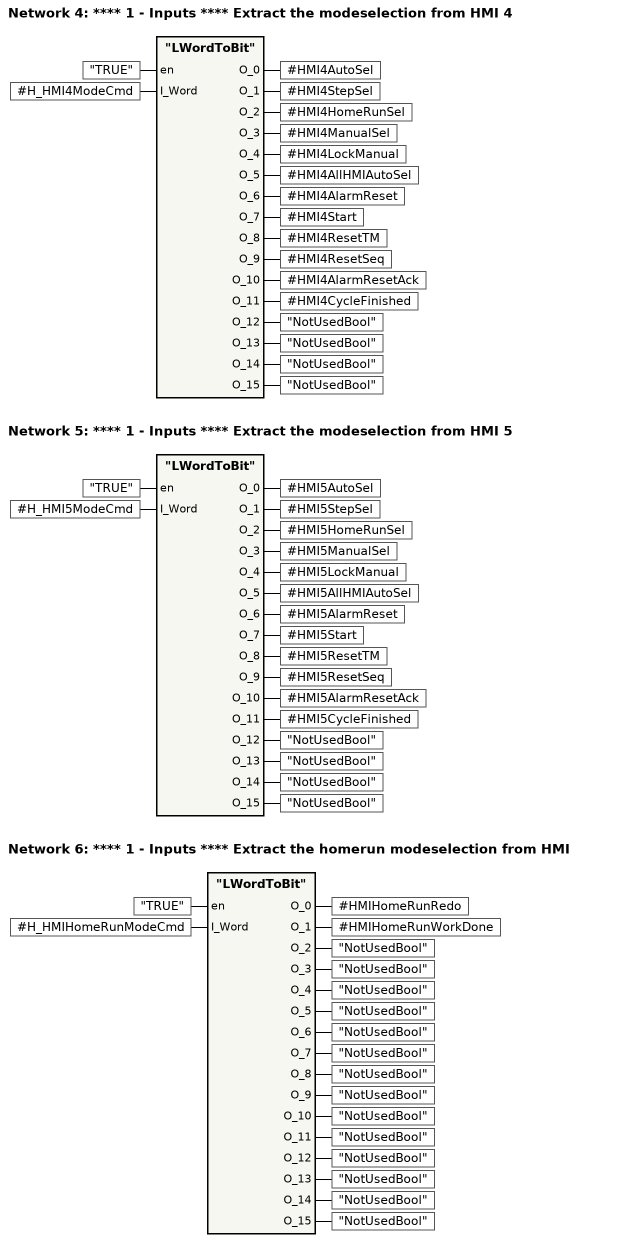
   IF "TRUE" THEN
       "LWordToBit"(I_Word := #H_HMI4ModeCmd,
                    O_0 => #HMI4AutoSel,
                    O_1 => #HMI4StepSel,
                    O_2 => #HMI4HomeRunSel,
                    O_3 => #HMI4ManualSel,
                    O_4 => #HMI4LockManual,
                    O_5 => #HMI4AllHMIAutoSel,
                    O_6 => #HMI4AlarmReset,
                    O_7 => #HMI4Start,
                    O_8 => #HMI4ResetTM,
                    O_9 => #HMI4ResetSeq,
                    O_10 => #HMI4AlarmResetAck,
                    O_11 => #HMI4CycleFinished,
                    O_12 => "NotUsedBool",
                    O_13 => "NotUsedBool",
                    O_14 => "NotUsedBool",
                    O_15 => "NotUsedBool");
   END_IF;
END_REGION

REGION Network 5: **** 1 - Inputs **** Extract the modeselection from HMI 5
   // Extract the modeselection from HMI 5
   IF "TRUE" THEN
       "LWordToBit"(I_Word := #H_HMI5ModeCmd,
                    O_0 => #HMI5AutoSel,
                    O_1 => #HMI5StepSel,
                    O_2 => #HMI5HomeRunSel,
                    O_3 => #HMI5ManualSel,
                    O_4 => #HMI5LockManual,
                    O_5 => #HMI5AllHMIAutoSel,
                    O_6 => #HMI5AlarmReset,
                    O_7 => #HMI5Start,
                    O_8 => #HMI5ResetTM,
                    O_9 => #HMI5ResetSeq,
                    O_10 => #HMI5AlarmResetAck,
                    O_11 => #HMI5CycleFinished,
                    O_12 => "NotUsedBool",
                    O_13 => "NotUsedBool",
                    O_14 => "NotUsedBool",
                    O_15 => "NotUsedBool");
   END_IF;
END_REGION

REGION Network 6: **** 1 - Inputs **** Extract the homerun modeselection from HMI
   // Extract the homerun modeselection from HMI
   IF "TRUE" THEN
       "LWordToBit"(I_Word := #H_HMIHomeRunModeCmd,
                    O_0 => #HMIHomeRunRedo,
                    O_1 => #HMIHomeRunWorkDone,
                    O_2 => "NotUsedBool",
                    O_3 => "NotUsedBool",
                    O_4 => "NotUsedBool",
                    O_5 => "NotUsedBool",
                    O_6 => "NotUsedBool",
                    O_7 => "NotUsedBool",
                    O_8 => "NotUsedBool",
                    O_9 => "NotUsedBool",
                    O_10 => "NotUsedBool",
                    O_11 => "NotUsedBool",
                    O_12 => "NotUsedBool",
                    O_13 => "NotUsedBool",
                    O_14 => "NotUsedBool",
                    O_15 => "NotUsedBool");
   END_IF;
END_REGION

REGION Network 7: **** 1 - Inputs **** All HMI Auto selected
   // All HMI Auto selected
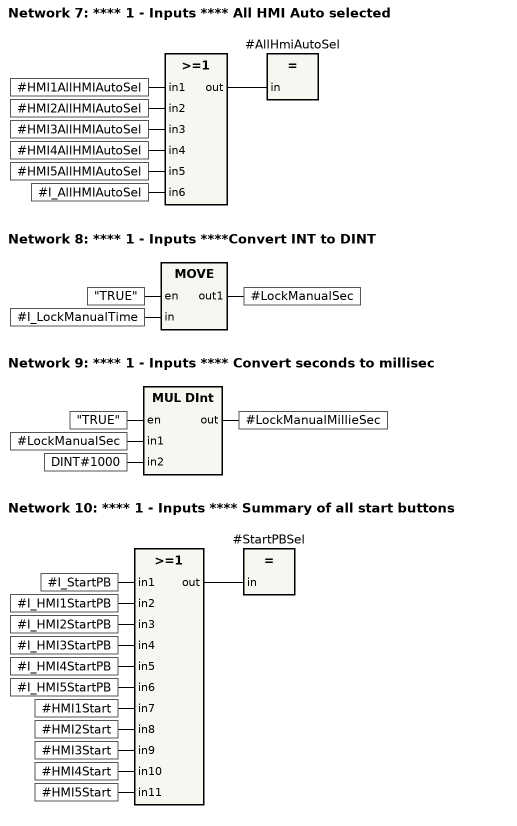
   #AllHmiAutoSel := #HMI1AllHMIAutoSel OR #HMI2AllHMIAutoSel OR #HMI3AllHMIAutoSel OR #HMI4AllHMIAutoSel OR #HMI5AllHMIAutoSel OR #I_AllHMIAutoSel;
END_REGION

REGION Network 8: **** 1 - Inputs ****Convert INT to DINT
   // Convert INT to DINT
   IF "TRUE" THEN #LockManualSec := #I_LockManualTime; END_IF;
END_REGION

REGION Network 9: **** 1 - Inputs **** Convert seconds to millisec
   // Convert seconds to millisec
   IF "TRUE" THEN #LockManualMillieSec := #LockManualSec * DINT#1000; END_IF;
END_REGION

REGION Network 10: **** 1 - Inputs **** Summary of all start buttons
   // Summary of all start buttons
   #StartPBSel := #I_StartPB OR #I_HMI1StartPB OR #I_HMI2StartPB OR #I_HMI3StartPB OR #I_HMI4StartPB OR #I_HMI5StartPB OR #HMI1Start OR #HMI2Start OR #HMI3Start OR #HMI4Start OR #HMI5Start;
END_REGION

REGION Network 11: **** 1 - Inputs **** Reset Start button from HMI
   // Reset Start button from HMI
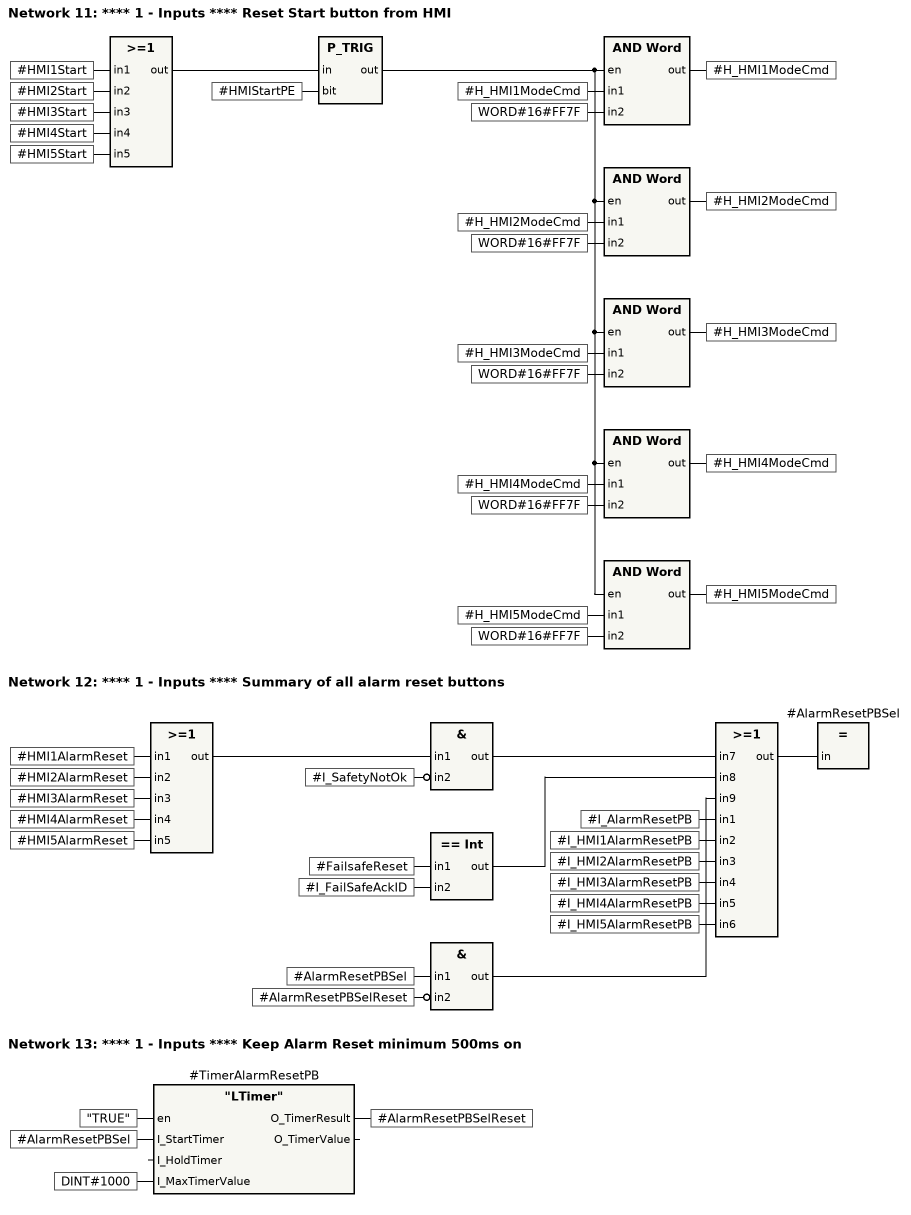
   #_w1 := #HMI1Start OR #HMI2Start OR #HMI3Start OR #HMI4Start OR #HMI5Start;
   #_w2 := #_w1 AND NOT #HMIStartPE;   // rising edge
   #HMIStartPE := #_w1;
   IF #_w2 THEN
       #H_HMI1ModeCmd := #H_HMI1ModeCmd AND WORD#16#FF7F;
       #H_HMI2ModeCmd := #H_HMI2ModeCmd AND WORD#16#FF7F;
       #H_HMI3ModeCmd := #H_HMI3ModeCmd AND WORD#16#FF7F;
       #H_HMI4ModeCmd := #H_HMI4ModeCmd AND WORD#16#FF7F;
       #H_HMI5ModeCmd := #H_HMI5ModeCmd AND WORD#16#FF7F;
   END_IF;
END_REGION

REGION Network 12: **** 1 - Inputs **** Summary of all alarm reset buttons
   // Summary of all alarm reset buttons
   #AlarmResetPBSel := ((#HMI1AlarmReset OR #HMI2AlarmReset OR #HMI3AlarmReset OR #HMI4AlarmReset OR #HMI5AlarmReset) AND NOT #I_SafetyNotOk) OR (#FailsafeReset = #I_FailSafeAckID) OR (#AlarmResetPBSel AND NOT #AlarmResetPBSelReset) OR #I_AlarmResetPB OR #I_HMI1AlarmResetPB OR #I_HMI2AlarmResetPB OR #I_HMI3AlarmResetPB OR #I_HMI4AlarmResetPB OR #I_HMI5AlarmResetPB;
END_REGION

REGION Network 13: **** 1 - Inputs **** Keep Alarm Reset minimum 500ms on
   // Keep Alarm Reset minimum 500ms on
   IF "TRUE" THEN
       #TimerAlarmResetPB(I_StartTimer := #AlarmResetPBSel,   // "LTimer"
                          I_MaxTimerValue := DINT#1000,
                          O_TimerResult => #AlarmResetPBSelReset);
   END_IF;
END_REGION

REGION Network 14: **** 1 - Inputs **** Reset AlarmResetPb from HMI
   // Reset AlarmResetPb from HMI
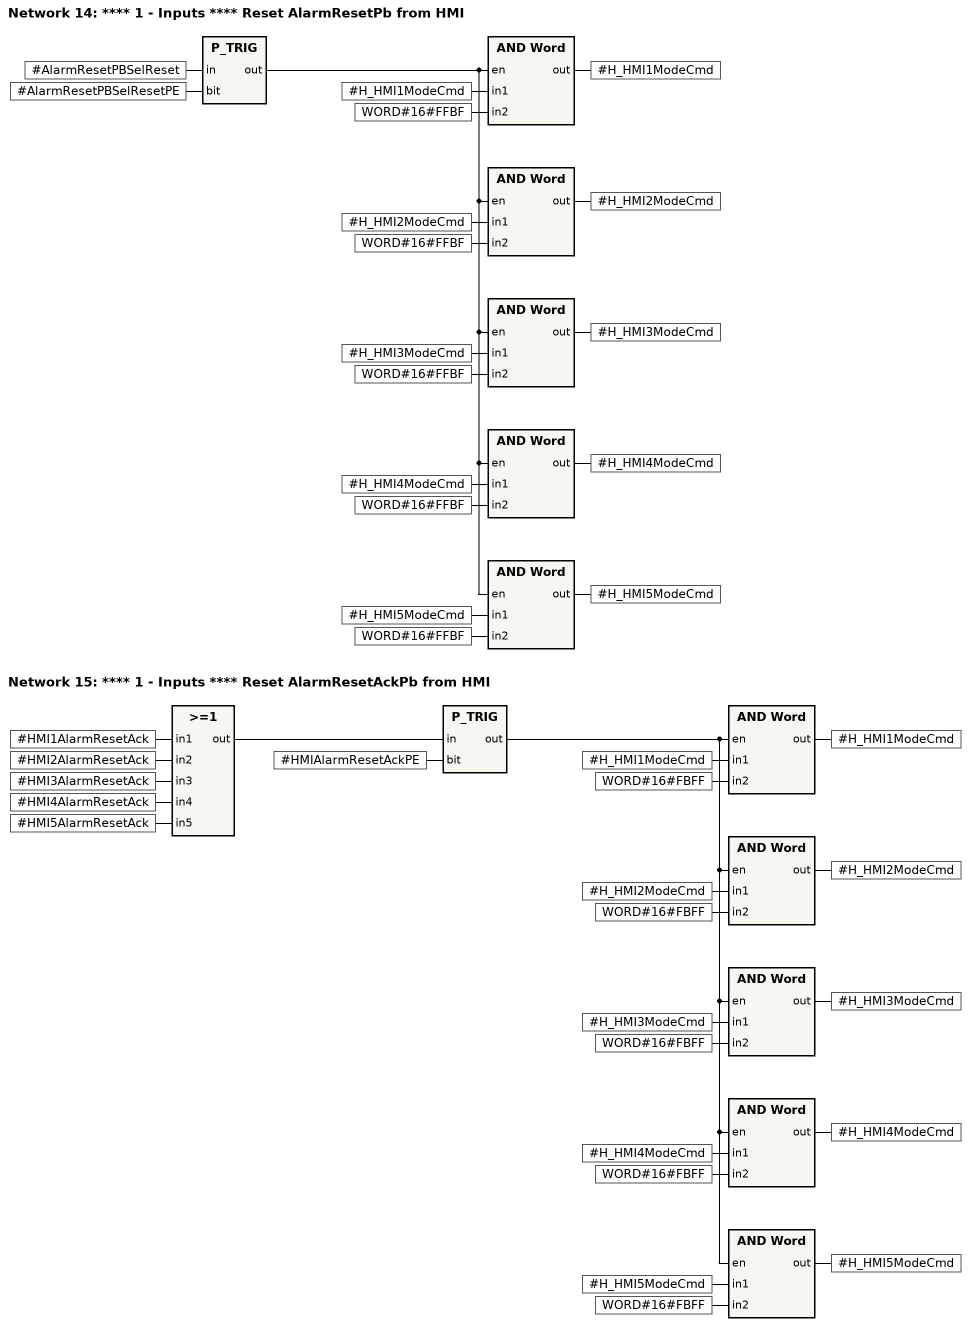
   #_w1 := #AlarmResetPBSelReset AND NOT #AlarmResetPBSelResetPE;   // rising edge
   #AlarmResetPBSelResetPE := #AlarmResetPBSelReset;
   IF #_w1 THEN
       #H_HMI1ModeCmd := #H_HMI1ModeCmd AND WORD#16#FFBF;
       #H_HMI2ModeCmd := #H_HMI2ModeCmd AND WORD#16#FFBF;
       #H_HMI3ModeCmd := #H_HMI3ModeCmd AND WORD#16#FFBF;
       #H_HMI4ModeCmd := #H_HMI4ModeCmd AND WORD#16#FFBF;
       #H_HMI5ModeCmd := #H_HMI5ModeCmd AND WORD#16#FFBF;
   END_IF;
END_REGION

REGION Network 15: **** 1 - Inputs **** Reset AlarmResetAckPb from HMI
   // Reset AlarmResetAckPb from HMI
   #_w1 := #HMI1AlarmResetAck OR #HMI2AlarmResetAck OR #HMI3AlarmResetAck OR #HMI4AlarmResetAck OR #HMI5AlarmResetAck;
   #_w2 := #_w1 AND NOT #HMIAlarmResetAckPE;   // rising edge
   #HMIAlarmResetAckPE := #_w1;
   IF #_w2 THEN
       #H_HMI1ModeCmd := #H_HMI1ModeCmd AND WORD#16#FBFF;
       #H_HMI2ModeCmd := #H_HMI2ModeCmd AND WORD#16#FBFF;
       #H_HMI3ModeCmd := #H_HMI3ModeCmd AND WORD#16#FBFF;
       #H_HMI4ModeCmd := #H_HMI4ModeCmd AND WORD#16#FBFF;
       #H_HMI5ModeCmd := #H_HMI5ModeCmd AND WORD#16#FBFF;
   END_IF;
END_REGION

REGION Network 16: **** 1 - Inputs **** Reset ResetTM button from HMI
   // Reset ResetTM button from HMI
